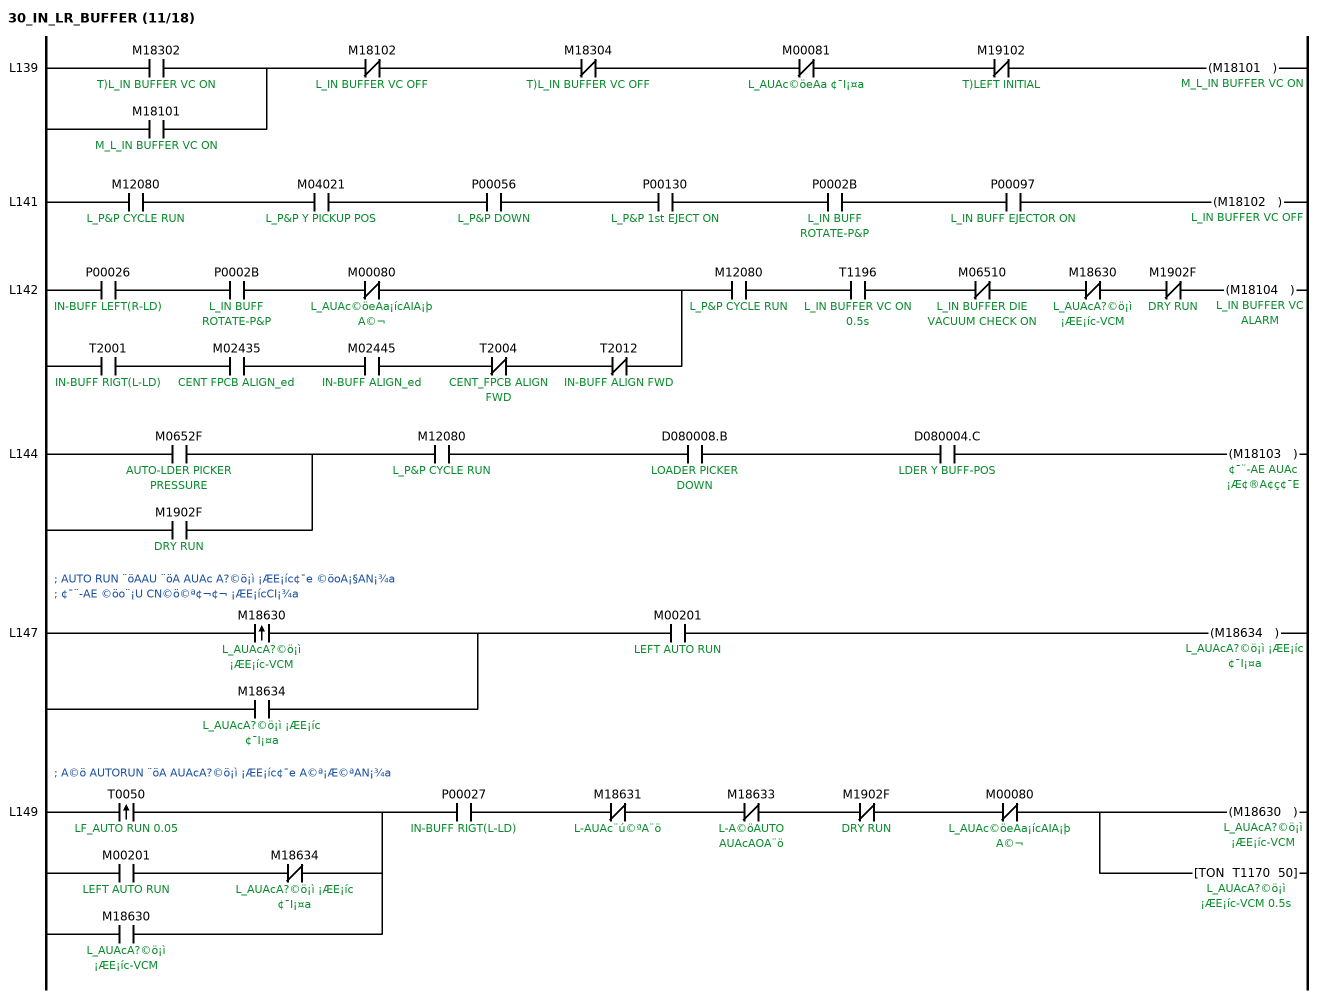
[picture p216: 30_IN_LR_BUFFER rungs L139-L149]
; L139
LOAD      M18302	// T)L_IN BUFFER VC ON
OR        M18101	// M_L_IN BUFFER VC ON
AND NOT   M18102	// L_IN BUFFER VC OFF
AND NOT   M18304	// T)L_IN BUFFER VC OFF
AND NOT   M00081	// L_AUAc©öeAa ¢¯I¡¤a
AND NOT   M19102	// T)LEFT INITIAL
OUT       M18101	// M_L_IN BUFFER VC ON
; L141
LOAD      M12080	// L_P&P CYCLE RUN
AND       M04021	// L_P&P Y PICKUP POS
AND       P00056	// L_P&P DOWN
AND       P00130	// L_P&P 1st EJECT ON
AND       P0002B	// L_IN BUFF ROTATE-P&P
AND       P00097	// L_IN BUFF EJECTOR ON
OUT       M18102	// L_IN BUFFER VC OFF
; L142
LOAD      P00026	// IN-BUFF LEFT(R-LD)
AND       P0002B	// L_IN BUFF ROTATE-P&P
AND NOT   M00080	// L_AUAc©öeAa¡ícAIA¡þA©¬
LOAD      T2001	// IN-BUFF RIGT(L-LD)
AND       M02435	// CENT FPCB ALIGN_ed
AND       M02445	// IN-BUFF ALIGN_ed
AND NOT   T2004	// CENT_FPCB ALIGN FWD
AND NOT   T2012	// IN-BUFF ALIGN FWD
OR LOAD
AND       M12080	// L_P&P CYCLE RUN
AND       T1196	// L_IN BUFFER VC ON 0.5s
AND NOT   M06510	// L_IN BUFFER DIE VACUUM CHECK ON
AND NOT   M18630	// L_AUAcA?©ö¡ì ¡ÆE¡íc-VCM
AND NOT   M1902F	// DRY RUN
OUT       M18104	// L_IN BUFFER VC ALARM
; L144
LOAD      M0652F	// AUTO-LDER PICKER PRESSURE
OR        M1902F	// DRY RUN
AND       M12080	// L_P&P CYCLE RUN
AND       D080008.B	// LOADER PICKER DOWN
AND       D080004.C	// LDER Y BUFF-POS
OUT       M18103	// ¢¯¨­AE AUAc ¡Æ¢®A¢ç¢¯E
// AUTO RUN ¨öAAU ¨öA AUAc A?©ö¡ì ¡ÆE¡íc¢¯e ©öoA¡§AN¡¾a
; L147
LOADP     M18630	// L_AUAcA?©ö¡ì ¡ÆE¡íc-VCM
OR        M18634	// L_AUAcA?©ö¡ì ¡ÆE¡íc ¢¯I¡¤a
AND       M00201	// LEFT AUTO RUN
OUT       M18634	// L_AUAcA?©ö¡ì ¡ÆE¡íc ¢¯I¡¤a
// output comment: ¢¯¨­AE ©öo¨¡U CN©ö©ª¢¬¢¬ ¡ÆE¡ícCI¡¾a
; L149
LOADP     T0050	// LF_AUTO RUN 0.05
LOAD      M00201	// LEFT AUTO RUN
AND NOT   M18634	// L_AUAcA?©ö¡ì ¡ÆE¡íc ¢¯I¡¤a
OR LOAD
OR        M18630	// L_AUAcA?©ö¡ì ¡ÆE¡íc-VCM
AND       P00027	// IN-BUFF RIGT(L-LD)
AND NOT   M18631	// L-AUAc¨ú©ªA¨ö
AND NOT   M18633	// L-A©öAUTO AUAcAOA¨ö
AND NOT   M1902F	// DRY RUN
AND NOT   M00080	// L_AUAc©öeAa¡ícAIA¡þA©¬
OUT       M18630	// L_AUAcA?©ö¡ì ¡ÆE¡íc-VCM
TON       T1170 50	// L_AUAcA?©ö¡ì ¡ÆE¡íc-VCM 0.5s
// output comment: A©ö AUTORUN ¨öA AUAcA?©ö¡ì ¡ÆE¡íc¢¯e A©ª¡Æ©ªAN¡¾a

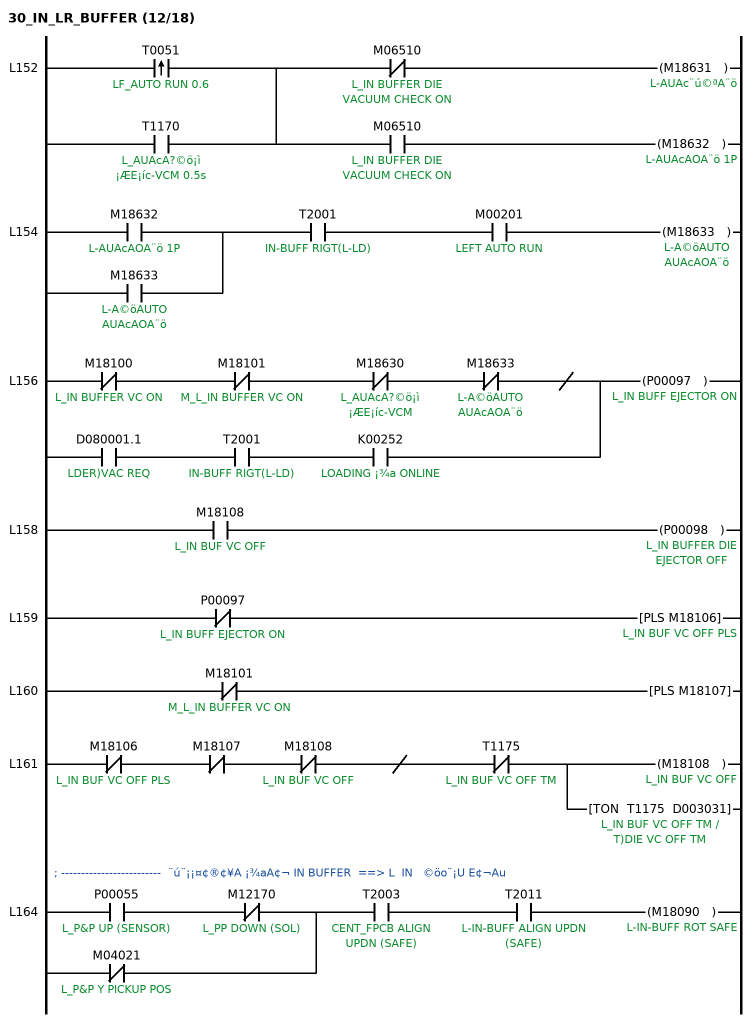
; L152
LOADP     T0051	// LF_AUTO RUN 0.6
OR        T1170	// L_AUAcA?©ö¡ì ¡ÆE¡íc-VCM 0.5s
MPUSH
AND NOT   M06510	// L_IN BUFFER DIE VACUUM CHECK ON
OUT       M18631	// L-AUAc¨ú©ªA¨ö
MPOP
AND       M06510	// L_IN BUFFER DIE VACUUM CHECK ON
OUT       M18632	// L-AUAcAOA¨ö 1P
; L154
LOAD      M18632	// L-AUAcAOA¨ö 1P
OR        M18633	// L-A©öAUTO AUAcAOA¨ö
AND       T2001	// IN-BUFF RIGT(L-LD)
AND       M00201	// LEFT AUTO RUN
OUT       M18633	// L-A©öAUTO AUAcAOA¨ö
; L156
LOAD NOT  M18100	// L_IN BUFFER VC ON
AND NOT   M18101	// M_L_IN BUFFER VC ON
AND NOT   M18630	// L_AUAcA?©ö¡ì ¡ÆE¡íc-VCM
AND NOT   M18633	// L-A©öAUTO AUAcAOA¨ö
NOT
LOAD      D080001.1	// LDER)VAC REQ
AND       T2001	// IN-BUFF RIGT(L-LD)
AND       K00252	// LOADING ¡¾a ONLINE
OR LOAD
OUT       P00097	// L_IN BUFF EJECTOR ON
; L158
LOAD      M18108	// L_IN BUF VC OFF
OUT       P00098	// L_IN BUFFER DIE EJECTOR OFF
; L159
LOAD NOT  P00097	// L_IN BUFF EJECTOR ON
OUTP      M18106	// L_IN BUF VC OFF PLS
; L160
LOAD NOT  M18101	// M_L_IN BUFFER VC ON
OUTP      M18107
; L161
LOAD NOT  M18106	// L_IN BUF VC OFF PLS
AND NOT   M18107
AND NOT   M18108	// L_IN BUF VC OFF
NOT
AND NOT   T1175	// L_IN BUF VC OFF TM
OUT       M18108	// L_IN BUF VC OFF
TON       T1175 D003031	// L_IN BUF VC OFF TM / T)DIE VC OFF TM
// -------------------------  ¨ú¨¡¡¤¢®¢¥A ¡¾aA¢¬ IN BUFFER  ==> L  IN   ©öo¨¡U E¢¬Au
; L164
LOAD      P00055	// L_P&P UP (SENSOR)
AND NOT   M12170	// L_PP DOWN (SOL)
OR NOT    M04021	// L_P&P Y PICKUP POS
AND       T2003	// CENT_FPCB ALIGN UPDN (SAFE)
AND       T2011	// L-IN-BUFF ALIGN UPDN (SAFE)
OUT       M18090	// L-IN-BUFF ROT SAFE

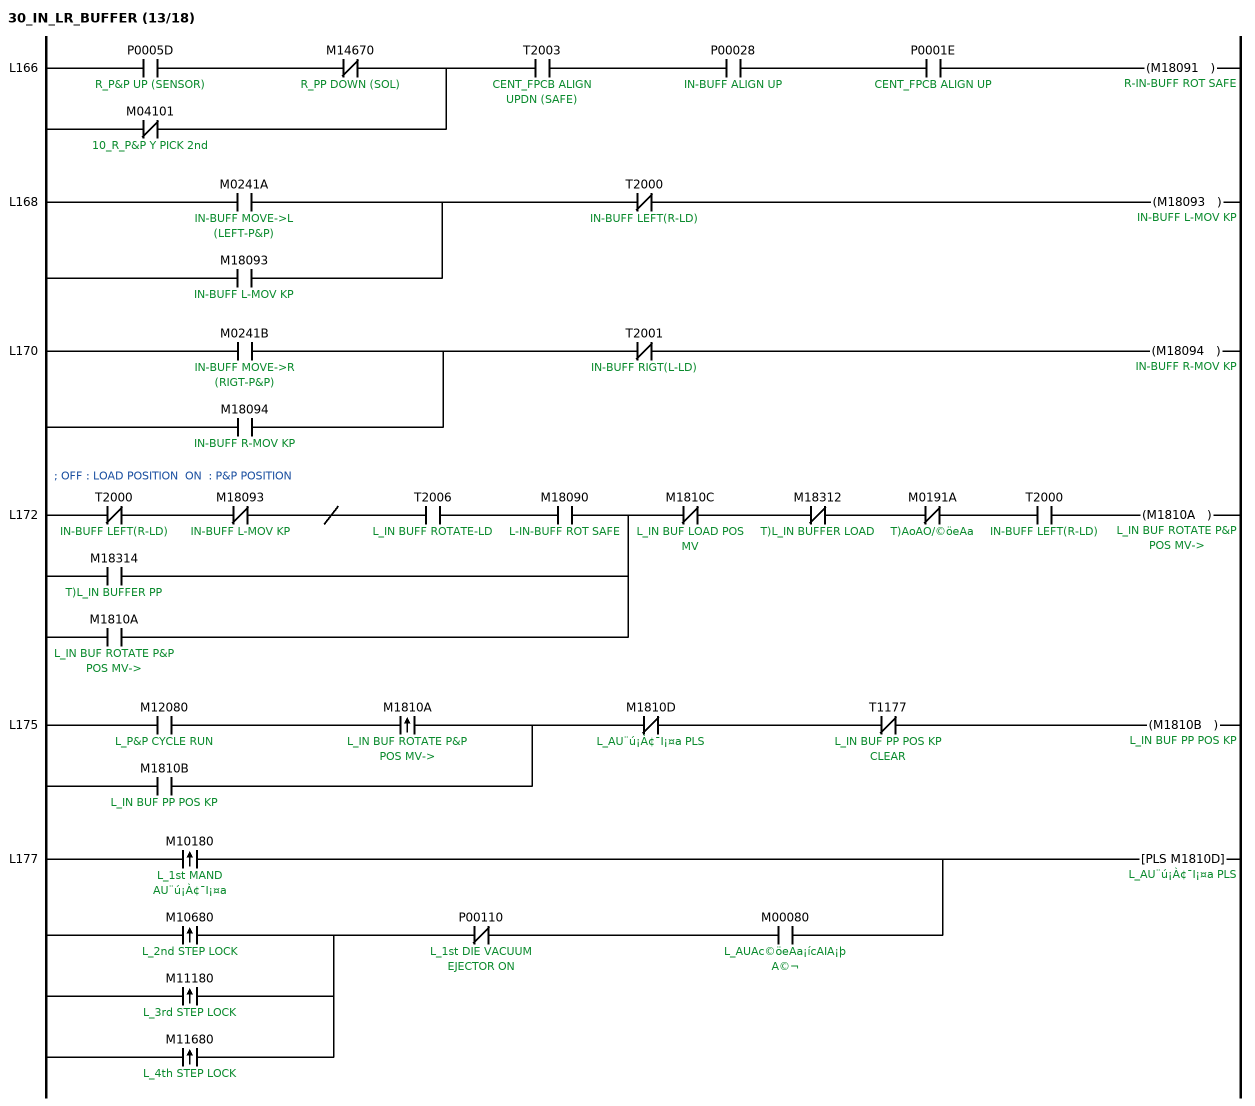
; L166
LOAD      P0005D	// R_P&P UP (SENSOR)
AND NOT   M14670	// R_PP DOWN (SOL)
OR NOT    M04101	// 10_R_P&P Y PICK 2nd
AND       T2003	// CENT_FPCB ALIGN UPDN (SAFE)
AND       P00028	// IN-BUFF ALIGN UP
AND       P0001E	// CENT_FPCB ALIGN UP
OUT       M18091	// R-IN-BUFF ROT SAFE
; L168
LOAD      M0241A	// IN-BUFF MOVE->L (LEFT-P&P)
OR        M18093	// IN-BUFF L-MOV KP
AND NOT   T2000	// IN-BUFF LEFT(R-LD)
OUT       M18093	// IN-BUFF L-MOV KP
; L170
LOAD      M0241B	// IN-BUFF MOVE->R (RIGT-P&P)
OR        M18094	// IN-BUFF R-MOV KP
AND NOT   T2001	// IN-BUFF RIGT(L-LD)
OUT       M18094	// IN-BUFF R-MOV KP
; L172
LOAD NOT  T2000	// IN-BUFF LEFT(R-LD)
AND NOT   M18093	// IN-BUFF L-MOV KP
NOT
AND       T2006	// L_IN BUFF ROTATE-LD
AND       M18090	// L-IN-BUFF ROT SAFE
OR        M18314	// T)L_IN BUFFER PP
OR        M1810A	// L_IN BUF ROTATE P&P POS MV->
AND NOT   M1810C	// L_IN BUF LOAD POS MV
AND NOT   M18312	// T)L_IN BUFFER LOAD
AND NOT   M0191A	// T)AoAO/©öeAa
AND       T2000	// IN-BUFF LEFT(R-LD)
OUT       M1810A	// L_IN BUF ROTATE P&P POS MV->
// output comment: OFF : LOAD POSITION  ON  : P&P POSITION
; L175
LOAD      M12080	// L_P&P CYCLE RUN
ANDP      M1810A	// L_IN BUF ROTATE P&P POS MV->
OR        M1810B	// L_IN BUF PP POS KP
AND NOT   M1810D	// L_AU¨ú¡À¢¯I¡¤a PLS
AND NOT   T1177	// L_IN BUF PP POS KP CLEAR
OUT       M1810B	// L_IN BUF PP POS KP
; L177
LOADP     M10180	// L_1st MAND AU¨ú¡À¢¯I¡¤a
LOADP     M10680	// L_2nd STEP LOCK
ORP       M11180	// L_3rd STEP LOCK
ORP       M11680	// L_4th STEP LOCK
AND NOT   P00110	// L_1st DIE VACUUM EJECTOR ON
AND       M00080	// L_AUAc©öeAa¡ícAIA¡þA©¬
OR LOAD
OUTP      M1810D	// L_AU¨ú¡À¢¯I¡¤a PLS

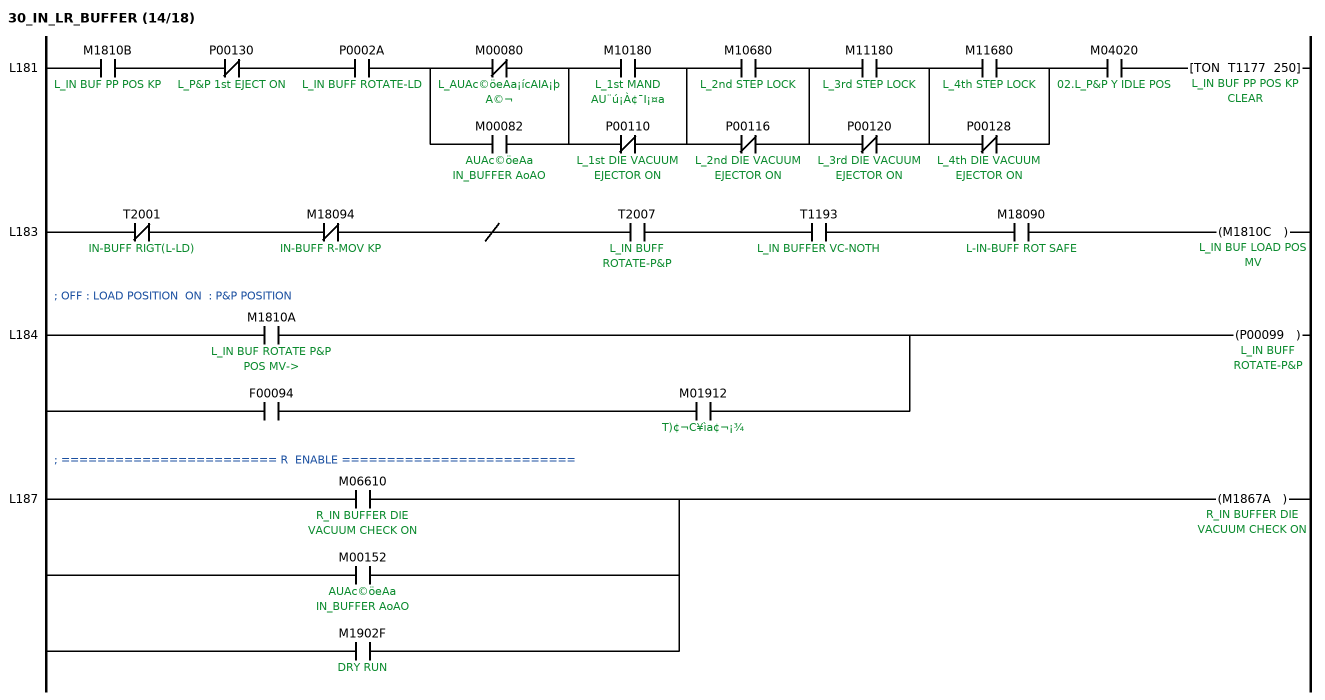
; L181
LOAD      M1810B	// L_IN BUF PP POS KP
AND NOT   P00130	// L_P&P 1st EJECT ON
AND       P0002A	// L_IN BUFF ROTATE-LD
LOAD NOT  M00080	// L_AUAc©öeAa¡ícAIA¡þA©¬
OR        M00082	// AUAc©öeAa IN_BUFFER AoAO 
AND LOAD
LOAD      M10180	// L_1st MAND AU¨ú¡À¢¯I¡¤a
OR NOT    P00110	// L_1st DIE VACUUM EJECTOR ON
AND LOAD
LOAD      M10680	// L_2nd STEP LOCK
OR NOT    P00116	// L_2nd DIE VACUUM EJECTOR ON
AND LOAD
LOAD      M11180	// L_3rd STEP LOCK
OR NOT    P00120	// L_3rd DIE VACUUM EJECTOR ON
AND LOAD
LOAD      M11680	// L_4th STEP LOCK
OR NOT    P00128	// L_4th DIE VACUUM EJECTOR ON
AND LOAD
AND       M04020	// 02.L_P&P Y IDLE POS
TON       T1177 250	// L_IN BUF PP POS KP CLEAR
; L183
LOAD NOT  T2001	// IN-BUFF RIGT(L-LD)
AND NOT   M18094	// IN-BUFF R-MOV KP
NOT
AND       T2007	// L_IN BUFF ROTATE-P&P
AND       T1193	// L_IN BUFFER VC-NOTH
AND       M18090	// L-IN-BUFF ROT SAFE
OUT       M1810C	// L_IN BUF LOAD POS MV
; L184
LOAD      M1810A	// L_IN BUF ROTATE P&P POS MV->
LOAD      F00094
AND       M01912	// T)¢¬C¥ìa¢¬¡¾
OR LOAD
OUT       P00099	// L_IN BUFF ROTATE-P&P
// output comment: OFF : LOAD POSITION  ON  : P&P POSITION
// ======================== R  ENABLE ==========================
; L187
LOAD      M06610	// R_IN BUFFER DIE VACUUM CHECK ON
OR        M00152	// AUAc©öeAa IN_BUFFER AoAO 
OR        M1902F	// DRY RUN
OUT       M1867A	// R_IN BUFFER DIE VACUUM CHECK ON

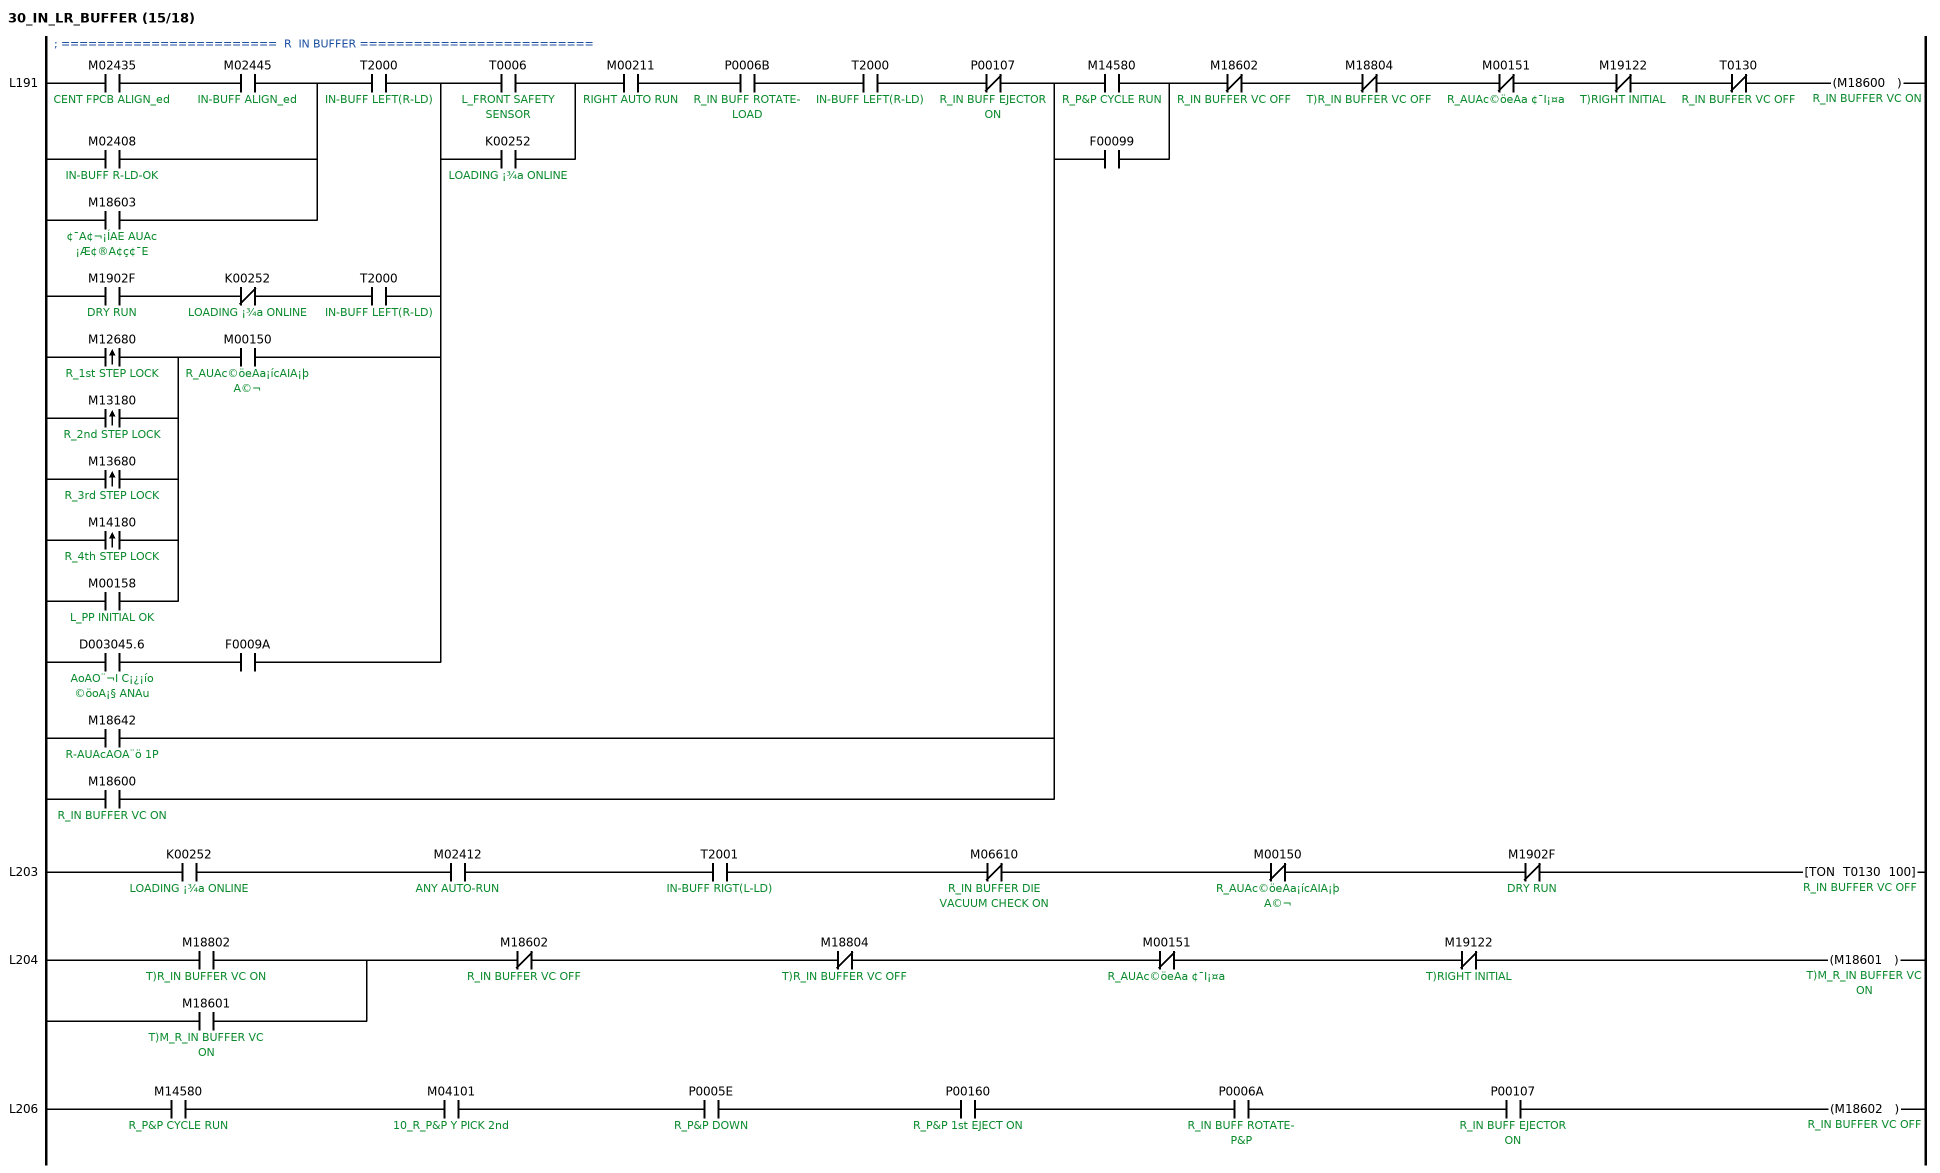
// ========================  R  IN BUFFER ==========================
; L191
LOAD      M02435	// CENT FPCB ALIGN_ed
AND       M02445	// IN-BUFF ALIGN_ed
OR        M02408	// IN-BUFF R-LD-OK
OR        M18603	// ¢¯A¢¬¡ÍAE AUAc ¡Æ¢®A¢ç¢¯E
AND       T2000	// IN-BUFF LEFT(R-LD)
LOAD      M1902F	// DRY RUN
AND NOT   K00252	// LOADING ¡¾a ONLINE
AND       T2000	// IN-BUFF LEFT(R-LD)
OR LOAD
LOADP     M12680	// R_1st STEP LOCK
ORP       M13180	// R_2nd STEP LOCK
ORP       M13680	// R_3rd STEP LOCK
ORP       M14180	// R_4th STEP LOCK
OR        M00158	// L_PP INITIAL OK
AND       M00150	// R_AUAc©öeAa¡ícAIA¡þA©¬
OR LOAD
LOAD      D003045.6	// AoAO¨¬I C¡¿¡ío ©öoA¡§ ANAu
AND       F0009A
OR LOAD
LOAD      T0006	// L_FRONT SAFETY SENSOR
OR        K00252	// LOADING ¡¾a ONLINE
AND LOAD
AND       M00211	// RIGHT AUTO RUN
AND       P0006B	// R_IN BUFF ROTATE- LOAD
AND       T2000	// IN-BUFF LEFT(R-LD)
AND NOT   P00107	// R_IN BUFF EJECTOR ON
OR        M18642	// R-AUAcAOA¨ö 1P
OR        M18600	// R_IN BUFFER VC ON
LOAD      M14580	// R_P&P CYCLE RUN
OR        F00099
AND LOAD
AND NOT   M18602	// R_IN BUFFER VC OFF
AND NOT   M18804	// T)R_IN BUFFER VC OFF
AND NOT   M00151	// R_AUAc©öeAa ¢¯I¡¤a
AND NOT   M19122	// T)RIGHT INITIAL
AND NOT   T0130	// R_IN BUFFER VC OFF
OUT       M18600	// R_IN BUFFER VC ON
; L203
LOAD      K00252	// LOADING ¡¾a ONLINE
AND       M02412	// ANY AUTO-RUN
AND       T2001	// IN-BUFF RIGT(L-LD)
AND NOT   M06610	// R_IN BUFFER DIE VACUUM CHECK ON
AND NOT   M00150	// R_AUAc©öeAa¡ícAIA¡þA©¬
AND NOT   M1902F	// DRY RUN
TON       T0130 100	// R_IN BUFFER VC OFF
; L204
LOAD      M18802	// T)R_IN BUFFER VC ON
OR        M18601	// T)M_R_IN BUFFER VC ON
AND NOT   M18602	// R_IN BUFFER VC OFF
AND NOT   M18804	// T)R_IN BUFFER VC OFF
AND NOT   M00151	// R_AUAc©öeAa ¢¯I¡¤a
AND NOT   M19122	// T)RIGHT INITIAL
OUT       M18601	// T)M_R_IN BUFFER VC ON
; L206
LOAD      M14580	// R_P&P CYCLE RUN
AND       M04101	// 10_R_P&P Y PICK 2nd
AND       P0005E	// R_P&P DOWN
AND       P00160	// R_P&P 1st EJECT ON
AND       P0006A	// R_IN BUFF ROTATE- P&P
AND       P00107	// R_IN BUFF EJECTOR ON
OUT       M18602	// R_IN BUFFER VC OFF

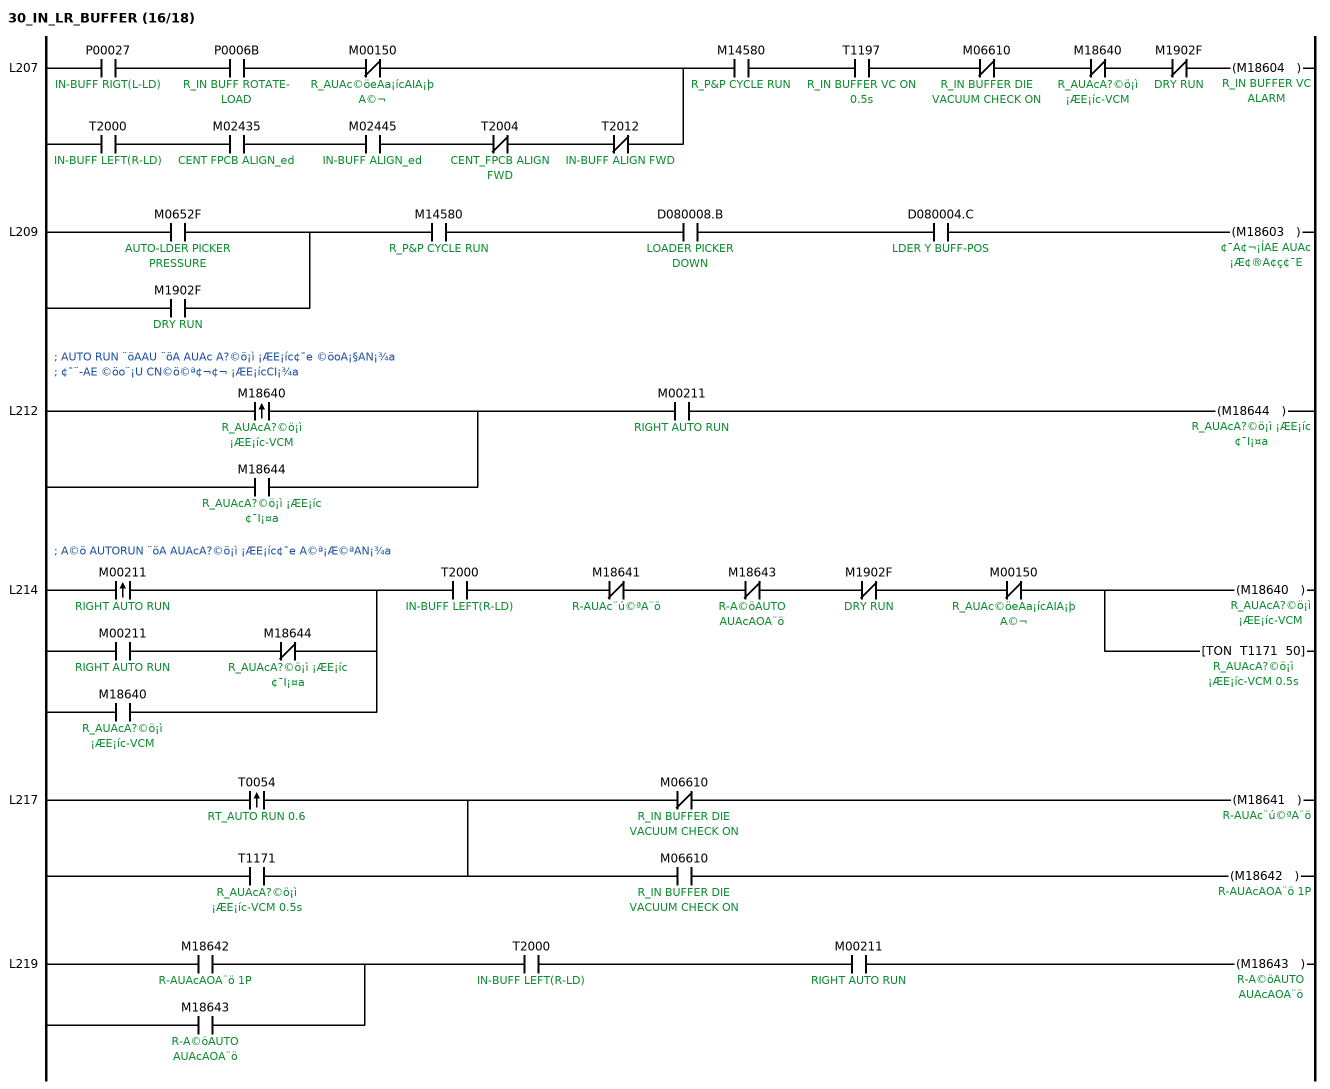
; L207
LOAD      P00027	// IN-BUFF RIGT(L-LD)
AND       P0006B	// R_IN BUFF ROTATE- LOAD
AND NOT   M00150	// R_AUAc©öeAa¡ícAIA¡þA©¬
LOAD      T2000	// IN-BUFF LEFT(R-LD)
AND       M02435	// CENT FPCB ALIGN_ed
AND       M02445	// IN-BUFF ALIGN_ed
AND NOT   T2004	// CENT_FPCB ALIGN FWD
AND NOT   T2012	// IN-BUFF ALIGN FWD
OR LOAD
AND       M14580	// R_P&P CYCLE RUN
AND       T1197	// R_IN BUFFER VC ON 0.5s
AND NOT   M06610	// R_IN BUFFER DIE VACUUM CHECK ON
AND NOT   M18640	// R_AUAcA?©ö¡ì ¡ÆE¡íc-VCM
AND NOT   M1902F	// DRY RUN
OUT       M18604	// R_IN BUFFER VC ALARM
; L209
LOAD      M0652F	// AUTO-LDER PICKER PRESSURE
OR        M1902F	// DRY RUN
AND       M14580	// R_P&P CYCLE RUN
AND       D080008.B	// LOADER PICKER DOWN
AND       D080004.C	// LDER Y BUFF-POS
OUT       M18603	// ¢¯A¢¬¡ÍAE AUAc ¡Æ¢®A¢ç¢¯E
// AUTO RUN ¨öAAU ¨öA AUAc A?©ö¡ì ¡ÆE¡íc¢¯e ©öoA¡§AN¡¾a
; L212
LOADP     M18640	// R_AUAcA?©ö¡ì ¡ÆE¡íc-VCM
OR        M18644	// R_AUAcA?©ö¡ì ¡ÆE¡íc ¢¯I¡¤a
AND       M00211	// RIGHT AUTO RUN
OUT       M18644	// R_AUAcA?©ö¡ì ¡ÆE¡íc ¢¯I¡¤a
// output comment: ¢¯¨­AE ©öo¨¡U CN©ö©ª¢¬¢¬ ¡ÆE¡ícCI¡¾a
; L214
LOADP     M00211	// RIGHT AUTO RUN
LOAD      M00211	// RIGHT AUTO RUN
AND NOT   M18644	// R_AUAcA?©ö¡ì ¡ÆE¡íc ¢¯I¡¤a
OR LOAD
OR        M18640	// R_AUAcA?©ö¡ì ¡ÆE¡íc-VCM
AND       T2000	// IN-BUFF LEFT(R-LD)
AND NOT   M18641	// R-AUAc¨ú©ªA¨ö
AND NOT   M18643	// R-A©öAUTO AUAcAOA¨ö
AND NOT   M1902F	// DRY RUN
AND NOT   M00150	// R_AUAc©öeAa¡ícAIA¡þA©¬
OUT       M18640	// R_AUAcA?©ö¡ì ¡ÆE¡íc-VCM
TON       T1171 50	// R_AUAcA?©ö¡ì ¡ÆE¡íc-VCM 0.5s
// output comment: A©ö AUTORUN ¨öA AUAcA?©ö¡ì ¡ÆE¡íc¢¯e A©ª¡Æ©ªAN¡¾a
; L217
LOADP     T0054	// RT_AUTO RUN 0.6
OR        T1171	// R_AUAcA?©ö¡ì ¡ÆE¡íc-VCM 0.5s
MPUSH
AND NOT   M06610	// R_IN BUFFER DIE VACUUM CHECK ON
OUT       M18641	// R-AUAc¨ú©ªA¨ö
MPOP
AND       M06610	// R_IN BUFFER DIE VACUUM CHECK ON
OUT       M18642	// R-AUAcAOA¨ö 1P
; L219
LOAD      M18642	// R-AUAcAOA¨ö 1P
OR        M18643	// R-A©öAUTO AUAcAOA¨ö
AND       T2000	// IN-BUFF LEFT(R-LD)
AND       M00211	// RIGHT AUTO RUN
OUT       M18643	// R-A©öAUTO AUAcAOA¨ö

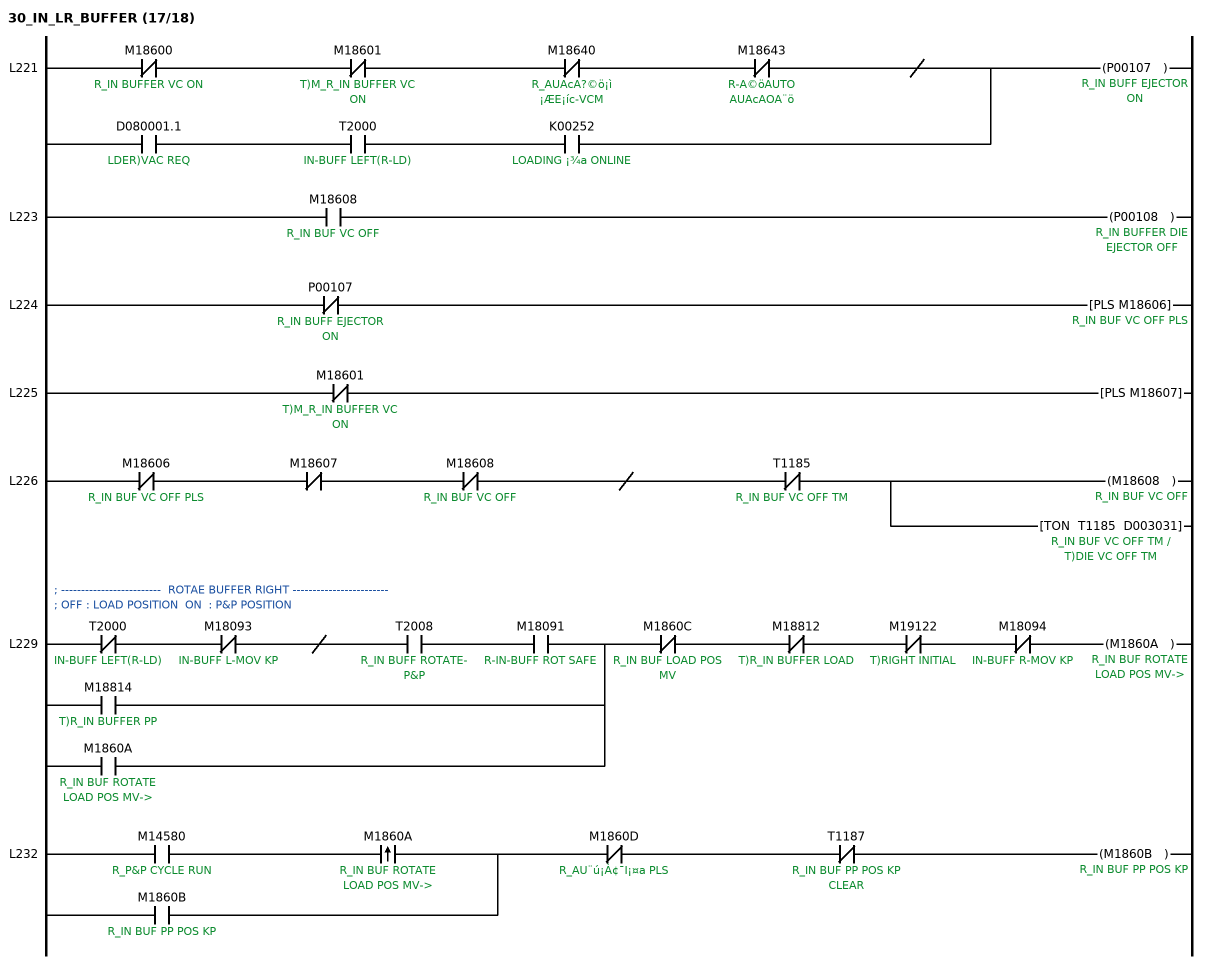
; L221
LOAD NOT  M18600	// R_IN BUFFER VC ON
AND NOT   M18601	// T)M_R_IN BUFFER VC ON
AND NOT   M18640	// R_AUAcA?©ö¡ì ¡ÆE¡íc-VCM
AND NOT   M18643	// R-A©öAUTO AUAcAOA¨ö
NOT
LOAD      D080001.1	// LDER)VAC REQ
AND       T2000	// IN-BUFF LEFT(R-LD)
AND       K00252	// LOADING ¡¾a ONLINE
OR LOAD
OUT       P00107	// R_IN BUFF EJECTOR ON
; L223
LOAD      M18608	// R_IN BUF VC OFF
OUT       P00108	// R_IN BUFFER DIE EJECTOR OFF
; L224
LOAD NOT  P00107	// R_IN BUFF EJECTOR ON
OUTP      M18606	// R_IN BUF VC OFF PLS
; L225
LOAD NOT  M18601	// T)M_R_IN BUFFER VC ON
OUTP      M18607
; L226
LOAD NOT  M18606	// R_IN BUF VC OFF PLS
AND NOT   M18607
AND NOT   M18608	// R_IN BUF VC OFF
NOT
AND NOT   T1185	// R_IN BUF VC OFF TM
OUT       M18608	// R_IN BUF VC OFF
TON       T1185 D003031	// R_IN BUF VC OFF TM / T)DIE VC OFF TM
// -------------------------  ROTAE BUFFER RIGHT ------------------------
; L229
LOAD NOT  T2000	// IN-BUFF LEFT(R-LD)
AND NOT   M18093	// IN-BUFF L-MOV KP
NOT
AND       T2008	// R_IN BUFF ROTATE- P&P
AND       M18091	// R-IN-BUFF ROT SAFE
OR        M18814	// T)R_IN BUFFER PP
OR        M1860A	// R_IN BUF ROTATE LOAD POS MV->
AND NOT   M1860C	// R_IN BUF LOAD POS MV
AND NOT   M18812	// T)R_IN BUFFER LOAD
AND NOT   M19122	// T)RIGHT INITIAL
AND NOT   M18094	// IN-BUFF R-MOV KP
OUT       M1860A	// R_IN BUF ROTATE LOAD POS MV->
// output comment: OFF : LOAD POSITION  ON  : P&P POSITION
; L232
LOAD      M14580	// R_P&P CYCLE RUN
ANDP      M1860A	// R_IN BUF ROTATE LOAD POS MV->
OR        M1860B	// R_IN BUF PP POS KP
AND NOT   M1860D	// R_AU¨ú¡À¢¯I¡¤a PLS
AND NOT   T1187	// R_IN BUF PP POS KP CLEAR
OUT       M1860B	// R_IN BUF PP POS KP

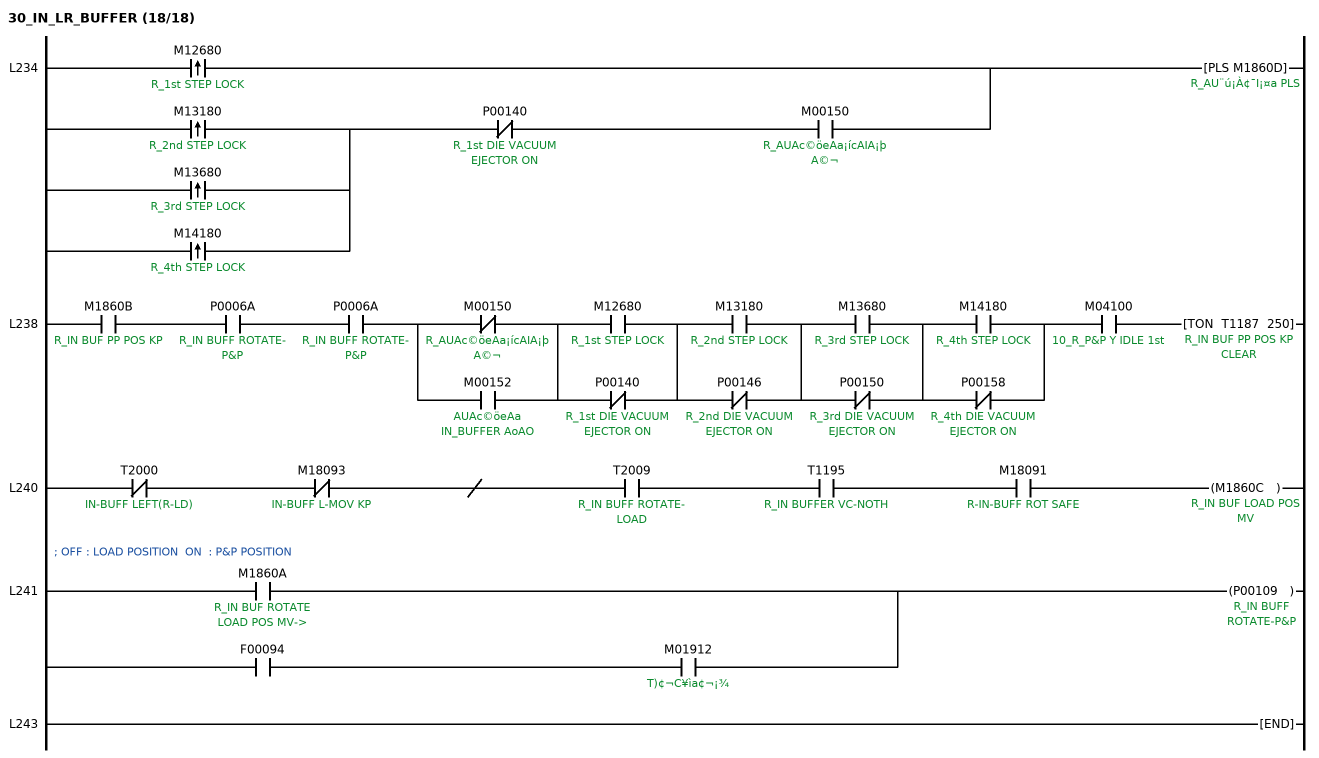
; L234
LOADP     M12680	// R_1st STEP LOCK
LOADP     M13180	// R_2nd STEP LOCK
ORP       M13680	// R_3rd STEP LOCK
ORP       M14180	// R_4th STEP LOCK
AND NOT   P00140	// R_1st DIE VACUUM EJECTOR ON
AND       M00150	// R_AUAc©öeAa¡ícAIA¡þA©¬
OR LOAD
OUTP      M1860D	// R_AU¨ú¡À¢¯I¡¤a PLS
; L238
LOAD      M1860B	// R_IN BUF PP POS KP
AND       P0006A	// R_IN BUFF ROTATE- P&P
AND       P0006A	// R_IN BUFF ROTATE- P&P
LOAD NOT  M00150	// R_AUAc©öeAa¡ícAIA¡þA©¬
OR        M00152	// AUAc©öeAa IN_BUFFER AoAO 
AND LOAD
LOAD      M12680	// R_1st STEP LOCK
OR NOT    P00140	// R_1st DIE VACUUM EJECTOR ON
AND LOAD
LOAD      M13180	// R_2nd STEP LOCK
OR NOT    P00146	// R_2nd DIE VACUUM EJECTOR ON
AND LOAD
LOAD      M13680	// R_3rd STEP LOCK
OR NOT    P00150	// R_3rd DIE VACUUM EJECTOR ON
AND LOAD
LOAD      M14180	// R_4th STEP LOCK
OR NOT    P00158	// R_4th DIE VACUUM EJECTOR ON
AND LOAD
AND       M04100	// 10_R_P&P Y IDLE 1st
TON       T1187 250	// R_IN BUF PP POS KP CLEAR
; L240
LOAD NOT  T2000	// IN-BUFF LEFT(R-LD)
AND NOT   M18093	// IN-BUFF L-MOV KP
NOT
AND       T2009	// R_IN BUFF ROTATE- LOAD
AND       T1195	// R_IN BUFFER VC-NOTH
AND       M18091	// R-IN-BUFF ROT SAFE
OUT       M1860C	// R_IN BUF LOAD POS MV
; L241
LOAD      M1860A	// R_IN BUF ROTATE LOAD POS MV->
LOAD      F00094
AND       M01912	// T)¢¬C¥ìa¢¬¡¾
OR LOAD
OUT       P00109	// R_IN BUFF ROTATE-P&P
// output comment: OFF : LOAD POSITION  ON  : P&P POSITION
; L243
END

PROGRAM 31_OUT_LR_BUFFER (task: ¨ö¨¬A¥ì CA¡¤I¡¾¡¿¡¤¡Í)

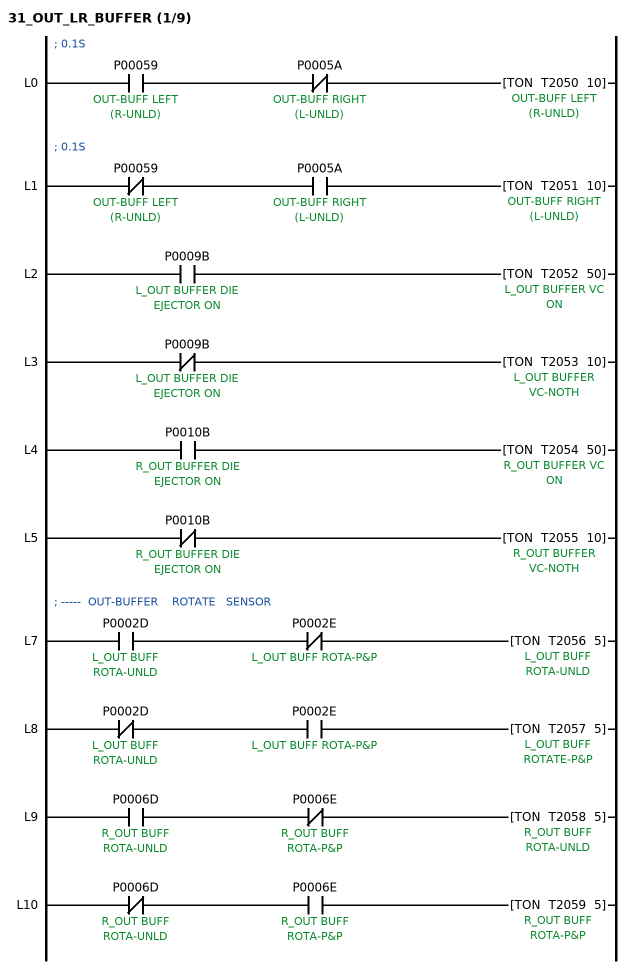
; L0
LOAD      P00059	// OUT-BUFF LEFT (R-UNLD)
AND NOT   P0005A	// OUT-BUFF RIGHT (L-UNLD)
TON       T2050 10	// OUT-BUFF LEFT (R-UNLD)
// output comment: 0.1S
; L1
LOAD NOT  P00059	// OUT-BUFF LEFT (R-UNLD)
AND       P0005A	// OUT-BUFF RIGHT (L-UNLD)
TON       T2051 10	// OUT-BUFF RIGHT (L-UNLD)
// output comment: 0.1S
; L2
LOAD      P0009B	// L_OUT BUFFER DIE EJECTOR ON
TON       T2052 50	// L_OUT BUFFER VC ON
; L3
LOAD NOT  P0009B	// L_OUT BUFFER DIE EJECTOR ON
TON       T2053 10	// L_OUT BUFFER VC-NOTH
; L4
LOAD      P0010B	// R_OUT BUFFER DIE EJECTOR ON
TON       T2054 50	// R_OUT BUFFER VC ON
; L5
LOAD NOT  P0010B	// R_OUT BUFFER DIE EJECTOR ON
TON       T2055 10	// R_OUT BUFFER VC-NOTH
// -----  OUT-BUFFER    ROTATE   SENSOR
; L7
LOAD      P0002D	// L_OUT BUFF ROTA-UNLD
AND NOT   P0002E	// L_OUT BUFF ROTA-P&P
TON       T2056 5	// L_OUT BUFF ROTA-UNLD
; L8
LOAD NOT  P0002D	// L_OUT BUFF ROTA-UNLD
AND       P0002E	// L_OUT BUFF ROTA-P&P
TON       T2057 5	// L_OUT BUFF ROTATE-P&P
; L9
LOAD      P0006D	// R_OUT BUFF ROTA-UNLD
AND NOT   P0006E	// R_OUT BUFF ROTA-P&P
TON       T2058 5	// R_OUT BUFF ROTA-UNLD
; L10
LOAD NOT  P0006D	// R_OUT BUFF ROTA-UNLD
AND       P0006E	// R_OUT BUFF ROTA-P&P
TON       T2059 5	// R_OUT BUFF ROTA-P&P

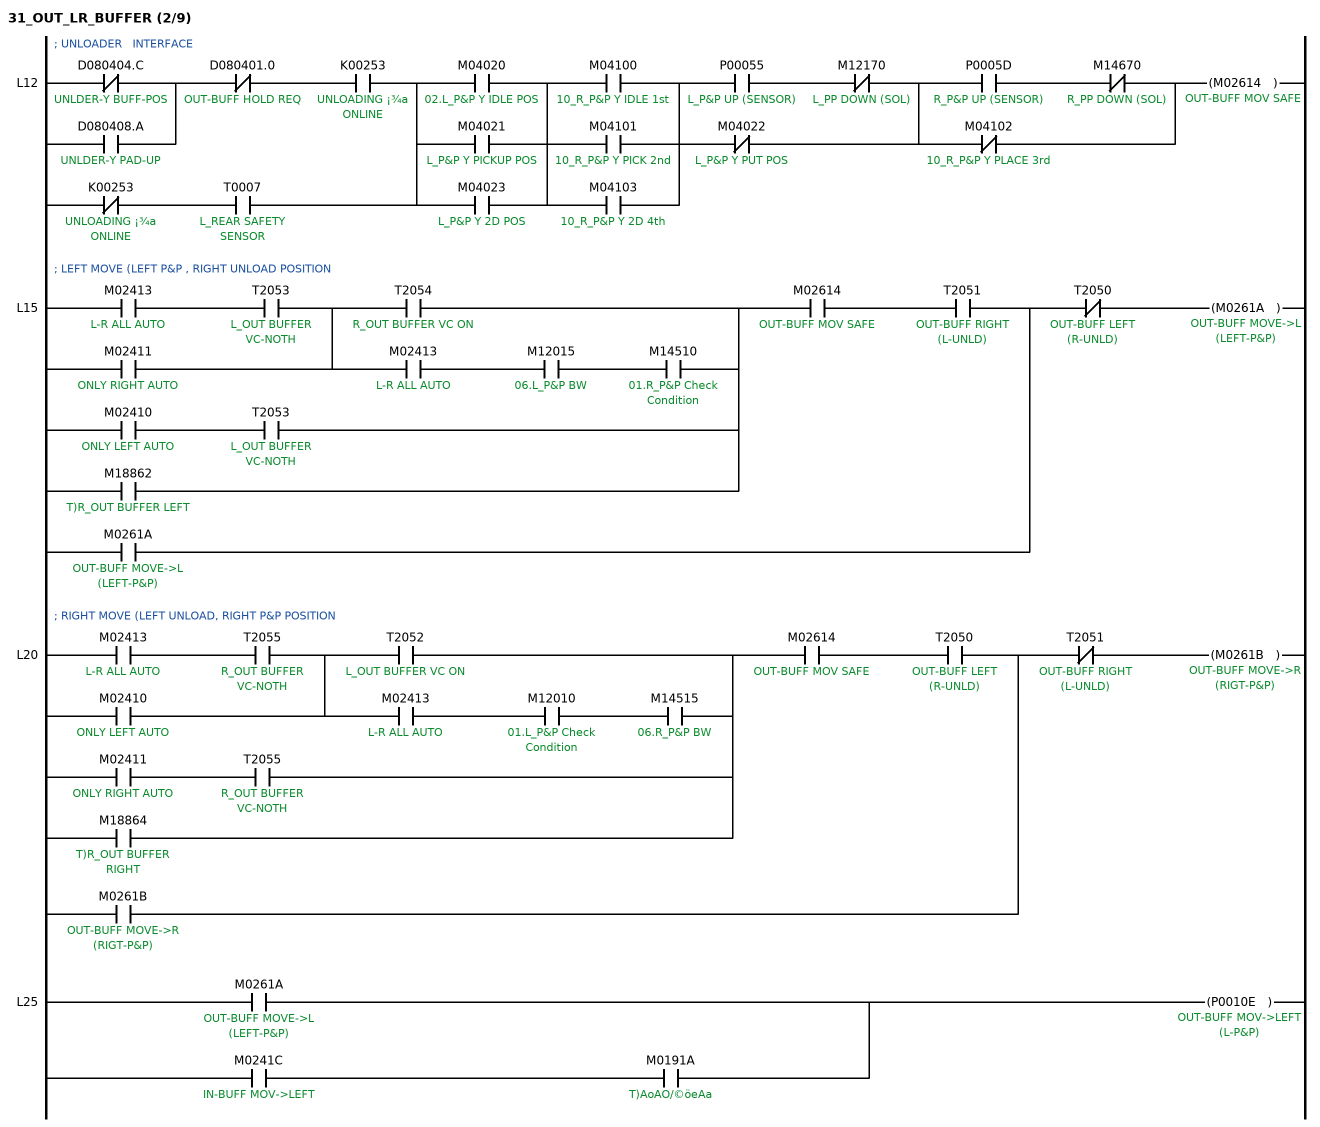
//  UNLOADER   INTERFACE
; L12
LOAD NOT  D080404.C	// UNLDER-Y BUFF-POS
OR        D080408.A	// UNLDER-Y PAD-UP
AND NOT   D080401.0	// OUT-BUFF HOLD REQ
AND       K00253	// UNLOADING ¡¾a ONLINE
LOAD NOT  K00253	// UNLOADING ¡¾a ONLINE
AND       T0007	// L_REAR SAFETY SENSOR
OR LOAD
LOAD      M04020	// 02.L_P&P Y IDLE POS
OR        M04021	// L_P&P Y PICKUP POS
OR        M04023	// L_P&P Y 2D POS
AND LOAD
LOAD      M04100	// 10_R_P&P Y IDLE 1st
OR        M04101	// 10_R_P&P Y PICK 2nd
OR        M04103	// 10_R_P&P Y 2D 4th
AND LOAD
LOAD      P00055	// L_P&P UP (SENSOR)
AND NOT   M12170	// L_PP DOWN (SOL)
OR NOT    M04022	// L_P&P Y PUT POS
AND LOAD
LOAD      P0005D	// R_P&P UP (SENSOR)
AND NOT   M14670	// R_PP DOWN (SOL)
OR NOT    M04102	// 10_R_P&P Y PLACE 3rd
AND LOAD
OUT       M02614	// OUT-BUFF MOV SAFE
; L15
LOAD      M02413	// L-R ALL AUTO
AND       T2053	// L_OUT BUFFER VC-NOTH
OR        M02411	// ONLY RIGHT AUTO
LOAD      T2054	// R_OUT BUFFER VC ON
LOAD      M02413	// L-R ALL AUTO
AND       M12015	// 06.L_P&P BW
AND       M14510	// 01.R_P&P Check Condition
OR LOAD
AND LOAD
LOAD      M02410	// ONLY LEFT AUTO
AND       T2053	// L_OUT BUFFER VC-NOTH
OR LOAD
OR        M18862	// T)R_OUT BUFFER LEFT
AND       M02614	// OUT-BUFF MOV SAFE
AND       T2051	// OUT-BUFF RIGHT (L-UNLD)
OR        M0261A	// OUT-BUFF MOVE->L (LEFT-P&P)
AND NOT   T2050	// OUT-BUFF LEFT (R-UNLD)
OUT       M0261A	// OUT-BUFF MOVE->L (LEFT-P&P)
// output comment: LEFT MOVE (LEFT P&P , RIGHT UNLOAD POSITION
; L20
LOAD      M02413	// L-R ALL AUTO
AND       T2055	// R_OUT BUFFER VC-NOTH
OR        M02410	// ONLY LEFT AUTO
LOAD      T2052	// L_OUT BUFFER VC ON
LOAD      M02413	// L-R ALL AUTO
AND       M12010	// 01.L_P&P Check Condition
AND       M14515	// 06.R_P&P BW
OR LOAD
AND LOAD
LOAD      M02411	// ONLY RIGHT AUTO
AND       T2055	// R_OUT BUFFER VC-NOTH
OR LOAD
OR        M18864	// T)R_OUT BUFFER RIGHT
AND       M02614	// OUT-BUFF MOV SAFE
AND       T2050	// OUT-BUFF LEFT (R-UNLD)
OR        M0261B	// OUT-BUFF MOVE->R (RIGT-P&P)
AND NOT   T2051	// OUT-BUFF RIGHT (L-UNLD)
OUT       M0261B	// OUT-BUFF MOVE->R (RIGT-P&P)
// output comment: RIGHT MOVE (LEFT UNLOAD, RIGHT P&P POSITION
; L25
LOAD      M0261A	// OUT-BUFF MOVE->L (LEFT-P&P)
LOAD      M0241C	// IN-BUFF MOV->LEFT
AND       M0191A	// T)AoAO/©öeAa
OR LOAD
OUT       P0010E	// OUT-BUFF MOV->LEFT (L-P&P)

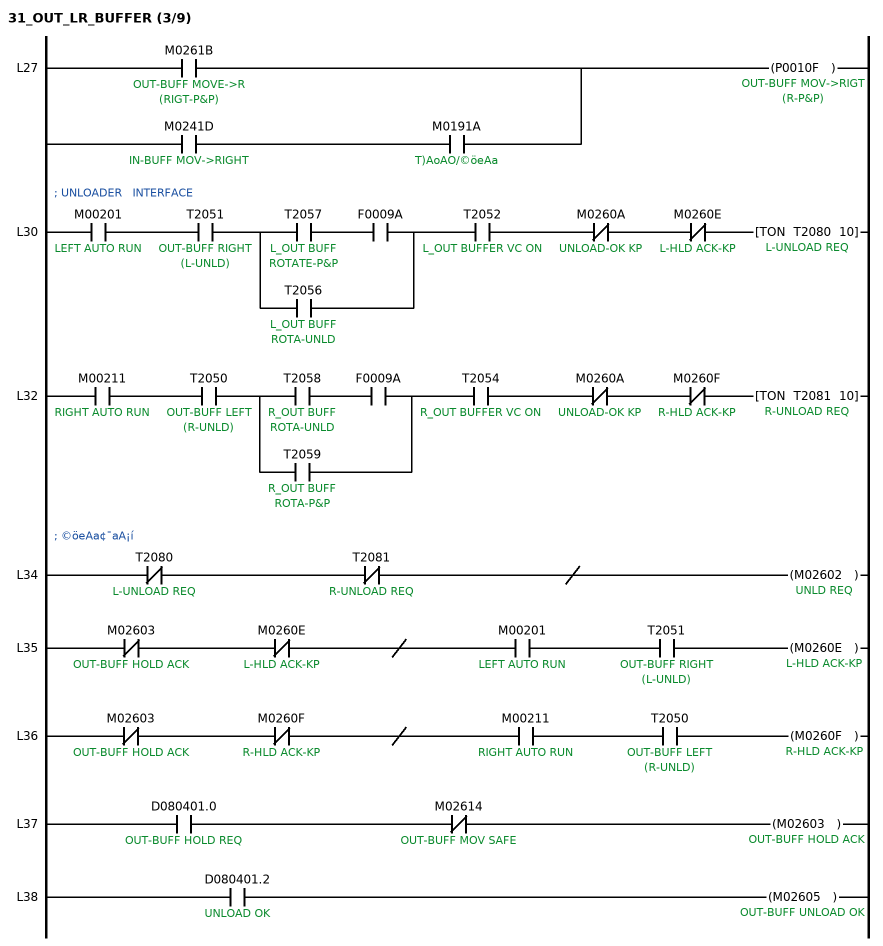
; L27
LOAD      M0261B	// OUT-BUFF MOVE->R (RIGT-P&P)
LOAD      M0241D	// IN-BUFF MOV->RIGHT
AND       M0191A	// T)AoAO/©öeAa
OR LOAD
OUT       P0010F	// OUT-BUFF MOV->RIGT (R-P&P)
//  UNLOADER   INTERFACE
; L30
LOAD      M00201	// LEFT AUTO RUN
AND       T2051	// OUT-BUFF RIGHT (L-UNLD)
LOAD      T2057	// L_OUT BUFF ROTATE-P&P
AND       F0009A
OR        T2056	// L_OUT BUFF ROTA-UNLD
AND LOAD
AND       T2052	// L_OUT BUFFER VC ON
AND NOT   M0260A	// UNLOAD-OK KP
AND NOT   M0260E	// L-HLD ACK-KP
TON       T2080 10	// L-UNLOAD REQ
; L32
LOAD      M00211	// RIGHT AUTO RUN
AND       T2050	// OUT-BUFF LEFT (R-UNLD)
LOAD      T2058	// R_OUT BUFF ROTA-UNLD
AND       F0009A
OR        T2059	// R_OUT BUFF ROTA-P&P
AND LOAD
AND       T2054	// R_OUT BUFFER VC ON
AND NOT   M0260A	// UNLOAD-OK KP
AND NOT   M0260F	// R-HLD ACK-KP
TON       T2081 10	// R-UNLOAD REQ
; L34
LOAD NOT  T2080	// L-UNLOAD REQ
AND NOT   T2081	// R-UNLOAD REQ
NOT
OUT       M02602	// UNLD REQ
// output comment: ©öeAa¢¯aA¡í
; L35
LOAD NOT  M02603	// OUT-BUFF HOLD ACK
AND NOT   M0260E	// L-HLD ACK-KP
NOT
AND       M00201	// LEFT AUTO RUN
AND       T2051	// OUT-BUFF RIGHT (L-UNLD)
OUT       M0260E	// L-HLD ACK-KP
; L36
LOAD NOT  M02603	// OUT-BUFF HOLD ACK
AND NOT   M0260F	// R-HLD ACK-KP
NOT
AND       M00211	// RIGHT AUTO RUN
AND       T2050	// OUT-BUFF LEFT (R-UNLD)
OUT       M0260F	// R-HLD ACK-KP
; L37
LOAD      D080401.0	// OUT-BUFF HOLD REQ
AND NOT   M02614	// OUT-BUFF MOV SAFE
OUT       M02603	// OUT-BUFF HOLD ACK
; L38
LOAD      D080401.2	// UNLOAD OK
OUT       M02605	// OUT-BUFF UNLOAD OK

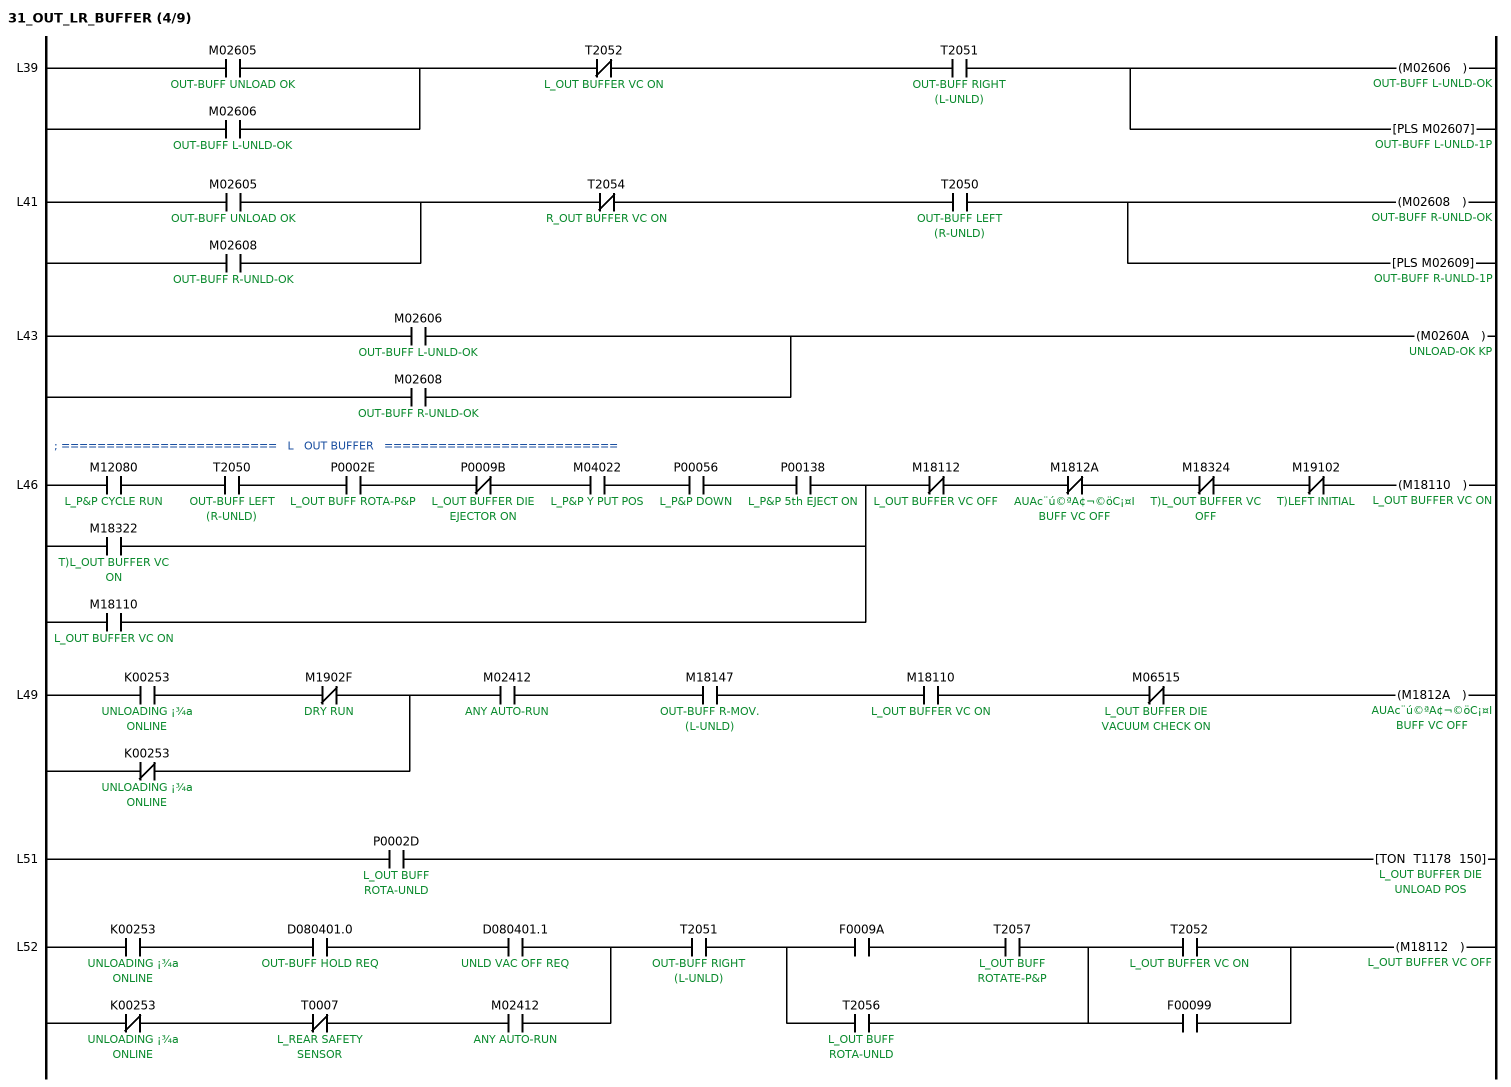
; L39
LOAD      M02605	// OUT-BUFF UNLOAD OK
OR        M02606	// OUT-BUFF L-UNLD-OK
AND NOT   T2052	// L_OUT BUFFER VC ON
AND       T2051	// OUT-BUFF RIGHT (L-UNLD)
OUT       M02606	// OUT-BUFF L-UNLD-OK
OUTP      M02607	// OUT-BUFF L-UNLD-1P
; L41
LOAD      M02605	// OUT-BUFF UNLOAD OK
OR        M02608	// OUT-BUFF R-UNLD-OK
AND NOT   T2054	// R_OUT BUFFER VC ON
AND       T2050	// OUT-BUFF LEFT (R-UNLD)
OUT       M02608	// OUT-BUFF R-UNLD-OK
OUTP      M02609	// OUT-BUFF R-UNLD-1P
; L43
LOAD      M02606	// OUT-BUFF L-UNLD-OK
OR        M02608	// OUT-BUFF R-UNLD-OK
OUT       M0260A	// UNLOAD-OK KP
// ========================   L   OUT BUFFER   ==========================
; L46
LOAD      M12080	// L_P&P CYCLE RUN
AND       T2050	// OUT-BUFF LEFT (R-UNLD)
AND       P0002E	// L_OUT BUFF ROTA-P&P
AND NOT   P0009B	// L_OUT BUFFER DIE EJECTOR ON
AND       M04022	// L_P&P Y PUT POS
AND       P00056	// L_P&P DOWN
AND       P00138	// L_P&P 5th EJECT ON
OR        M18322	// T)L_OUT BUFFER VC ON
OR        M18110	// L_OUT BUFFER VC ON
AND NOT   M18112	// L_OUT BUFFER VC OFF
AND NOT   M1812A	// AUAc¨ú©ªA¢¬©öC¡¤I BUFF VC OFF
AND NOT   M18324	// T)L_OUT BUFFER VC OFF
AND NOT   M19102	// T)LEFT INITIAL
OUT       M18110	// L_OUT BUFFER VC ON
; L49
LOAD      K00253	// UNLOADING ¡¾a ONLINE
AND NOT   M1902F	// DRY RUN
OR NOT    K00253	// UNLOADING ¡¾a ONLINE
AND       M02412	// ANY AUTO-RUN
AND       M18147	// OUT-BUFF R-MOV.  (L-UNLD)
AND       M18110	// L_OUT BUFFER VC ON
AND NOT   M06515	// L_OUT BUFFER DIE VACUUM CHECK ON
OUT       M1812A	// AUAc¨ú©ªA¢¬©öC¡¤I BUFF VC OFF
; L51
LOAD      P0002D	// L_OUT BUFF ROTA-UNLD
TON       T1178 150	// L_OUT BUFFER DIE UNLOAD POS
; L52
LOAD      K00253	// UNLOADING ¡¾a ONLINE
AND       D080401.0	// OUT-BUFF HOLD REQ
AND       D080401.1	// UNLD VAC OFF REQ
LOAD NOT  K00253	// UNLOADING ¡¾a ONLINE
AND NOT   T0007	// L_REAR SAFETY SENSOR
AND       M02412	// ANY AUTO-RUN
OR LOAD
AND       T2051	// OUT-BUFF RIGHT (L-UNLD)
LOAD      F0009A
AND       T2057	// L_OUT BUFF ROTATE-P&P
OR        T2056	// L_OUT BUFF ROTA-UNLD
AND LOAD
LOAD      T2052	// L_OUT BUFFER VC ON
OR        F00099
AND LOAD
OUT       M18112	// L_OUT BUFFER VC OFF

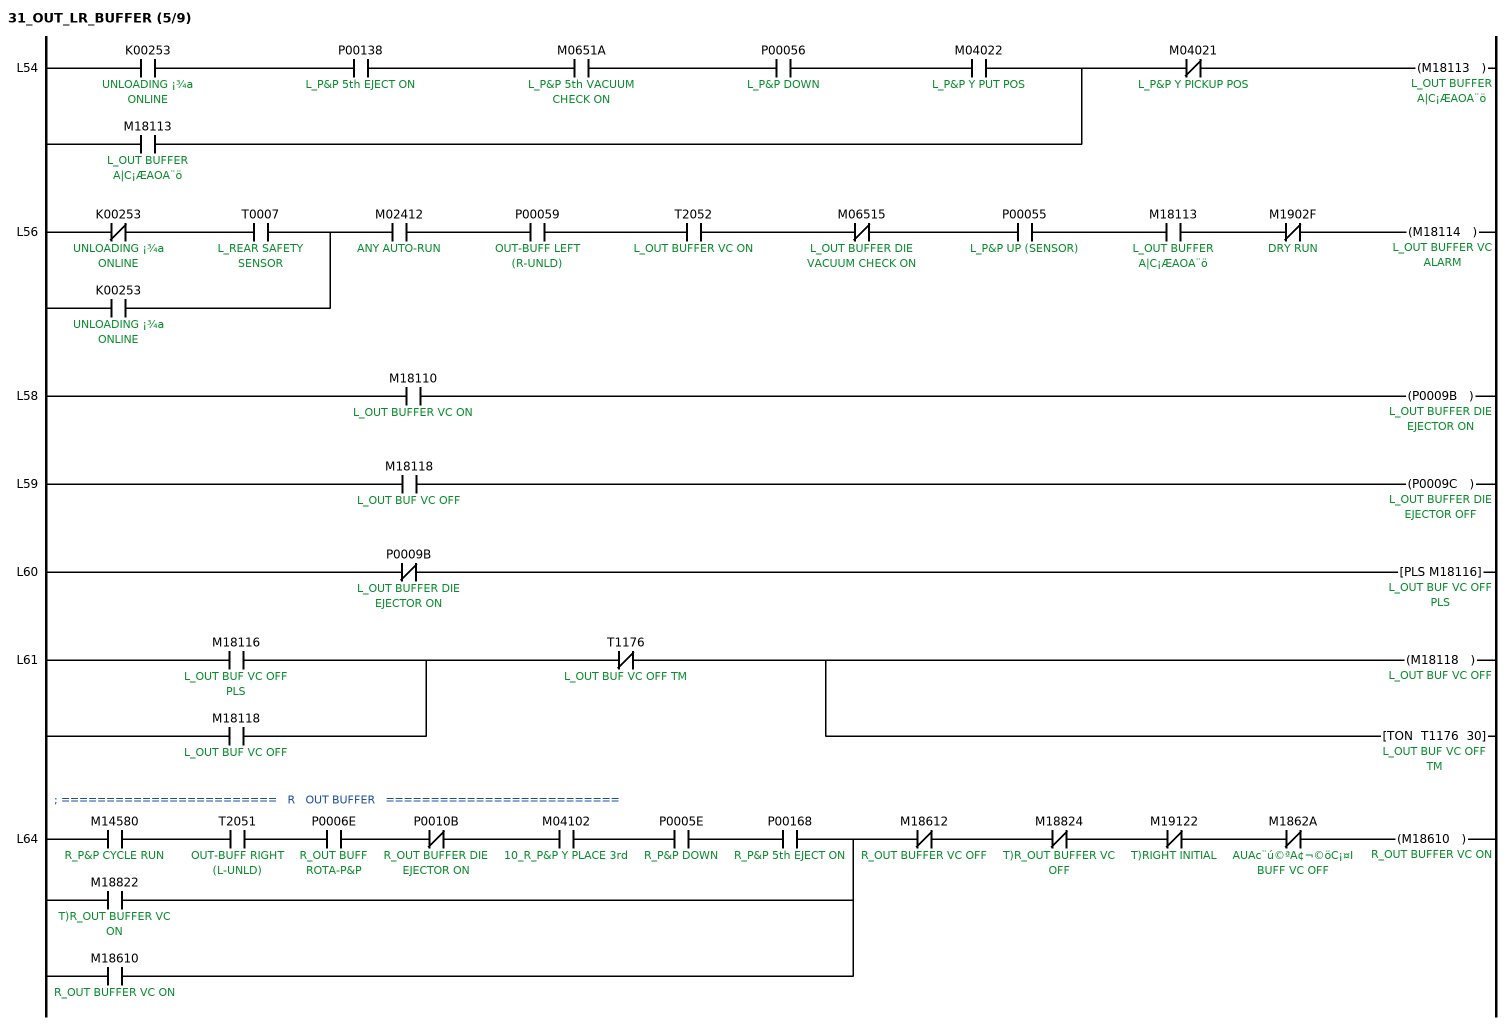
; L54
LOAD      K00253	// UNLOADING ¡¾a ONLINE
AND       P00138	// L_P&P 5th EJECT ON
AND       M0651A	// L_P&P 5th VACUUM CHECK ON
AND       P00056	// L_P&P DOWN
AND       M04022	// L_P&P Y PUT POS
OR        M18113	// L_OUT BUFFER A|C¡ÆAOA¨ö
AND NOT   M04021	// L_P&P Y PICKUP POS
OUT       M18113	// L_OUT BUFFER A|C¡ÆAOA¨ö
; L56
LOAD NOT  K00253	// UNLOADING ¡¾a ONLINE
AND       T0007	// L_REAR SAFETY SENSOR
OR        K00253	// UNLOADING ¡¾a ONLINE
AND       M02412	// ANY AUTO-RUN
AND       P00059	// OUT-BUFF LEFT (R-UNLD)
AND       T2052	// L_OUT BUFFER VC ON
AND NOT   M06515	// L_OUT BUFFER DIE VACUUM CHECK ON
AND       P00055	// L_P&P UP (SENSOR)
AND       M18113	// L_OUT BUFFER A|C¡ÆAOA¨ö
AND NOT   M1902F	// DRY RUN
OUT       M18114	// L_OUT BUFFER VC ALARM
; L58
LOAD      M18110	// L_OUT BUFFER VC ON
OUT       P0009B	// L_OUT BUFFER DIE EJECTOR ON
; L59
LOAD      M18118	// L_OUT BUF VC OFF
OUT       P0009C	// L_OUT BUFFER DIE EJECTOR OFF
; L60
LOAD NOT  P0009B	// L_OUT BUFFER DIE EJECTOR ON
OUTP      M18116	// L_OUT BUF VC OFF PLS
; L61
LOAD      M18116	// L_OUT BUF VC OFF PLS
OR        M18118	// L_OUT BUF VC OFF
AND NOT   T1176	// L_OUT BUF VC OFF TM
OUT       M18118	// L_OUT BUF VC OFF
TON       T1176 30	// L_OUT BUF VC OFF TM
// ========================   R   OUT BUFFER   ==========================
; L64
LOAD      M14580	// R_P&P CYCLE RUN
AND       T2051	// OUT-BUFF RIGHT (L-UNLD)
AND       P0006E	// R_OUT BUFF ROTA-P&P
AND NOT   P0010B	// R_OUT BUFFER DIE EJECTOR ON
AND       M04102	// 10_R_P&P Y PLACE 3rd
AND       P0005E	// R_P&P DOWN
AND       P00168	// R_P&P 5th EJECT ON
OR        M18822	// T)R_OUT BUFFER VC ON
OR        M18610	// R_OUT BUFFER VC ON
AND NOT   M18612	// R_OUT BUFFER VC OFF
AND NOT   M18824	// T)R_OUT BUFFER VC OFF
AND NOT   M19122	// T)RIGHT INITIAL
AND NOT   M1862A	// AUAc¨ú©ªA¢¬©öC¡¤I BUFF VC OFF
OUT       M18610	// R_OUT BUFFER VC ON

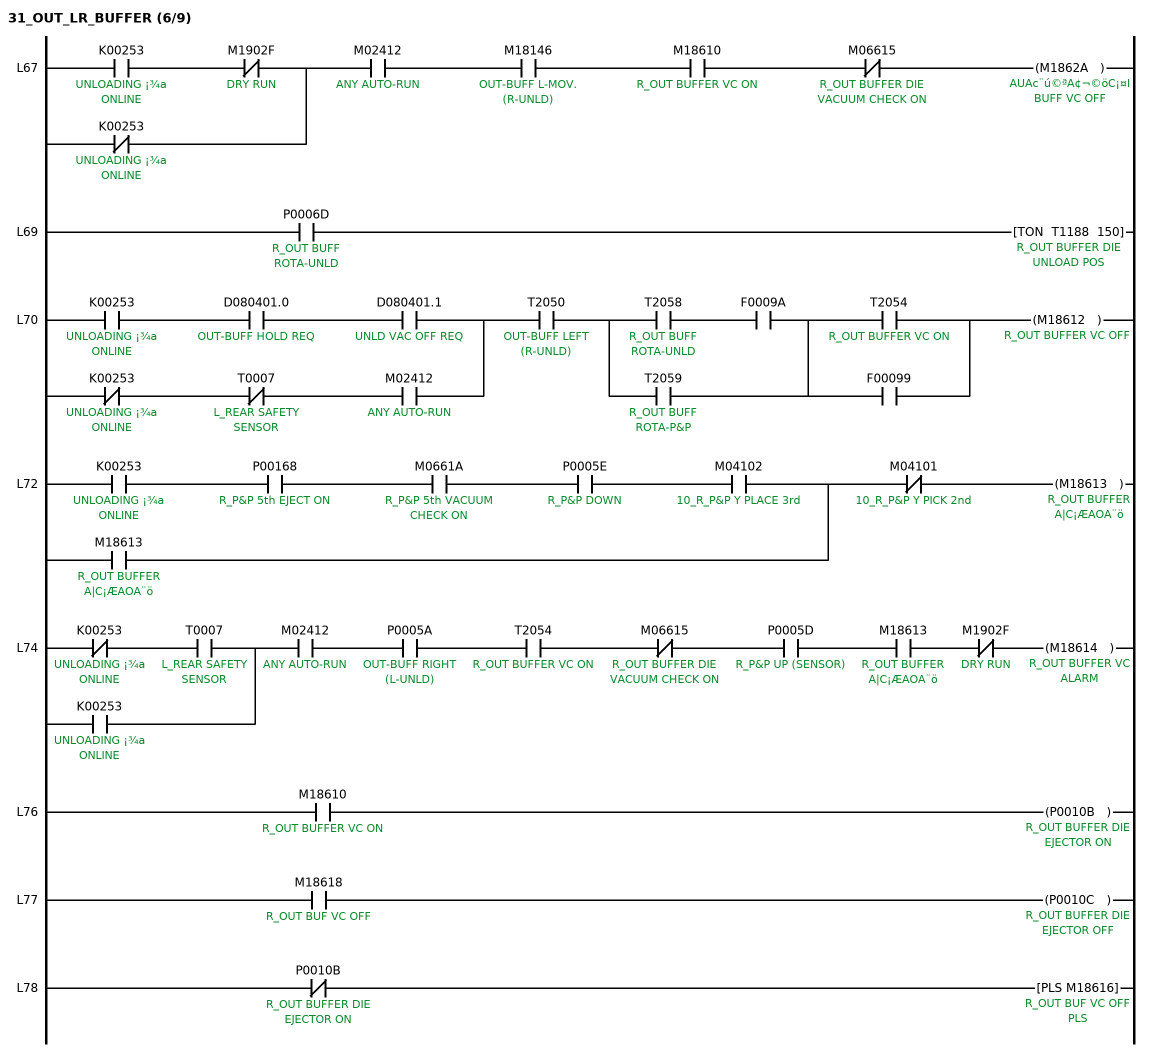
; L67
LOAD      K00253	// UNLOADING ¡¾a ONLINE
AND NOT   M1902F	// DRY RUN
OR NOT    K00253	// UNLOADING ¡¾a ONLINE
AND       M02412	// ANY AUTO-RUN
AND       M18146	// OUT-BUFF L-MOV.  (R-UNLD)
AND       M18610	// R_OUT BUFFER VC ON
AND NOT   M06615	// R_OUT BUFFER DIE VACUUM CHECK ON
OUT       M1862A	// AUAc¨ú©ªA¢¬©öC¡¤I BUFF VC OFF
; L69
LOAD      P0006D	// R_OUT BUFF ROTA-UNLD
TON       T1188 150	// R_OUT BUFFER DIE UNLOAD POS
; L70
LOAD      K00253	// UNLOADING ¡¾a ONLINE
AND       D080401.0	// OUT-BUFF HOLD REQ
AND       D080401.1	// UNLD VAC OFF REQ
LOAD NOT  K00253	// UNLOADING ¡¾a ONLINE
AND NOT   T0007	// L_REAR SAFETY SENSOR
AND       M02412	// ANY AUTO-RUN
OR LOAD
AND       T2050	// OUT-BUFF LEFT (R-UNLD)
LOAD      T2058	// R_OUT BUFF ROTA-UNLD
AND       F0009A
OR        T2059	// R_OUT BUFF ROTA-P&P
AND LOAD
LOAD      T2054	// R_OUT BUFFER VC ON
OR        F00099
AND LOAD
OUT       M18612	// R_OUT BUFFER VC OFF
; L72
LOAD      K00253	// UNLOADING ¡¾a ONLINE
AND       P00168	// R_P&P 5th EJECT ON
AND       M0661A	// R_P&P 5th VACUUM CHECK ON
AND       P0005E	// R_P&P DOWN
AND       M04102	// 10_R_P&P Y PLACE 3rd
OR        M18613	// R_OUT BUFFER A|C¡ÆAOA¨ö
AND NOT   M04101	// 10_R_P&P Y PICK 2nd
OUT       M18613	// R_OUT BUFFER A|C¡ÆAOA¨ö
; L74
LOAD NOT  K00253	// UNLOADING ¡¾a ONLINE
AND       T0007	// L_REAR SAFETY SENSOR
OR        K00253	// UNLOADING ¡¾a ONLINE
AND       M02412	// ANY AUTO-RUN
AND       P0005A	// OUT-BUFF RIGHT (L-UNLD)
AND       T2054	// R_OUT BUFFER VC ON
AND NOT   M06615	// R_OUT BUFFER DIE VACUUM CHECK ON
AND       P0005D	// R_P&P UP (SENSOR)
AND       M18613	// R_OUT BUFFER A|C¡ÆAOA¨ö
AND NOT   M1902F	// DRY RUN
OUT       M18614	// R_OUT BUFFER VC ALARM
; L76
LOAD      M18610	// R_OUT BUFFER VC ON
OUT       P0010B	// R_OUT BUFFER DIE EJECTOR ON
; L77
LOAD      M18618	// R_OUT BUF VC OFF
OUT       P0010C	// R_OUT BUFFER DIE EJECTOR OFF
; L78
LOAD NOT  P0010B	// R_OUT BUFFER DIE EJECTOR ON
OUTP      M18616	// R_OUT BUF VC OFF PLS

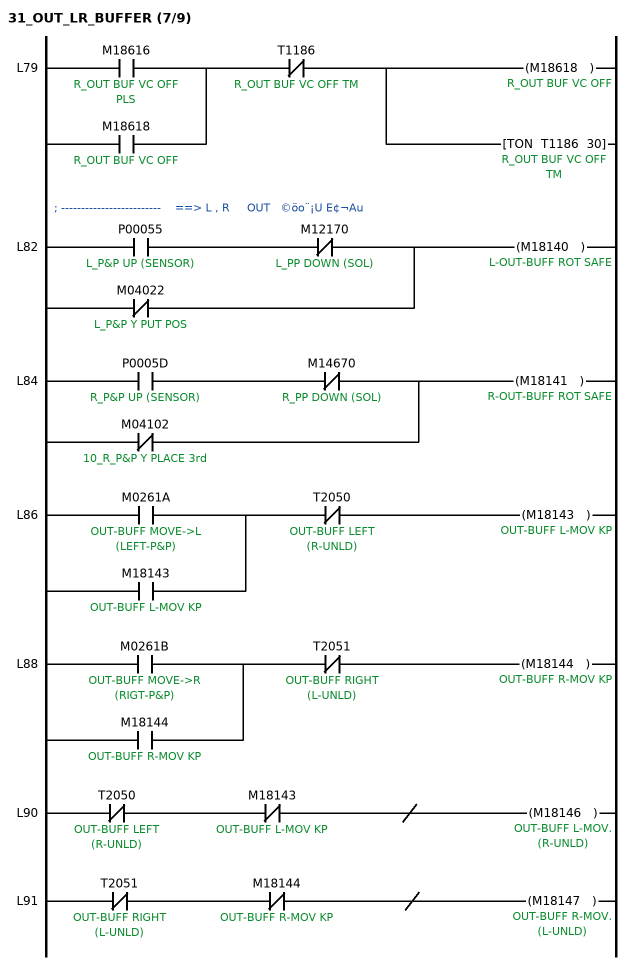
; L79
LOAD      M18616	// R_OUT BUF VC OFF PLS
OR        M18618	// R_OUT BUF VC OFF
AND NOT   T1186	// R_OUT BUF VC OFF TM
OUT       M18618	// R_OUT BUF VC OFF
TON       T1186 30	// R_OUT BUF VC OFF TM
// -------------------------    ==> L , R     OUT   ©öo¨¡U E¢¬Au
; L82
LOAD      P00055	// L_P&P UP (SENSOR)
AND NOT   M12170	// L_PP DOWN (SOL)
OR NOT    M04022	// L_P&P Y PUT POS
OUT       M18140	// L-OUT-BUFF ROT SAFE
; L84
LOAD      P0005D	// R_P&P UP (SENSOR)
AND NOT   M14670	// R_PP DOWN (SOL)
OR NOT    M04102	// 10_R_P&P Y PLACE 3rd
OUT       M18141	// R-OUT-BUFF ROT SAFE
; L86
LOAD      M0261A	// OUT-BUFF MOVE->L (LEFT-P&P)
OR        M18143	// OUT-BUFF L-MOV KP
AND NOT   T2050	// OUT-BUFF LEFT (R-UNLD)
OUT       M18143	// OUT-BUFF L-MOV KP
; L88
LOAD      M0261B	// OUT-BUFF MOVE->R (RIGT-P&P)
OR        M18144	// OUT-BUFF R-MOV KP
AND NOT   T2051	// OUT-BUFF RIGHT (L-UNLD)
OUT       M18144	// OUT-BUFF R-MOV KP
; L90
LOAD NOT  T2050	// OUT-BUFF LEFT (R-UNLD)
AND NOT   M18143	// OUT-BUFF L-MOV KP
NOT
OUT       M18146	// OUT-BUFF L-MOV.  (R-UNLD)
; L91
LOAD NOT  T2051	// OUT-BUFF RIGHT (L-UNLD)
AND NOT   M18144	// OUT-BUFF R-MOV KP
NOT
OUT       M18147	// OUT-BUFF R-MOV.  (L-UNLD)

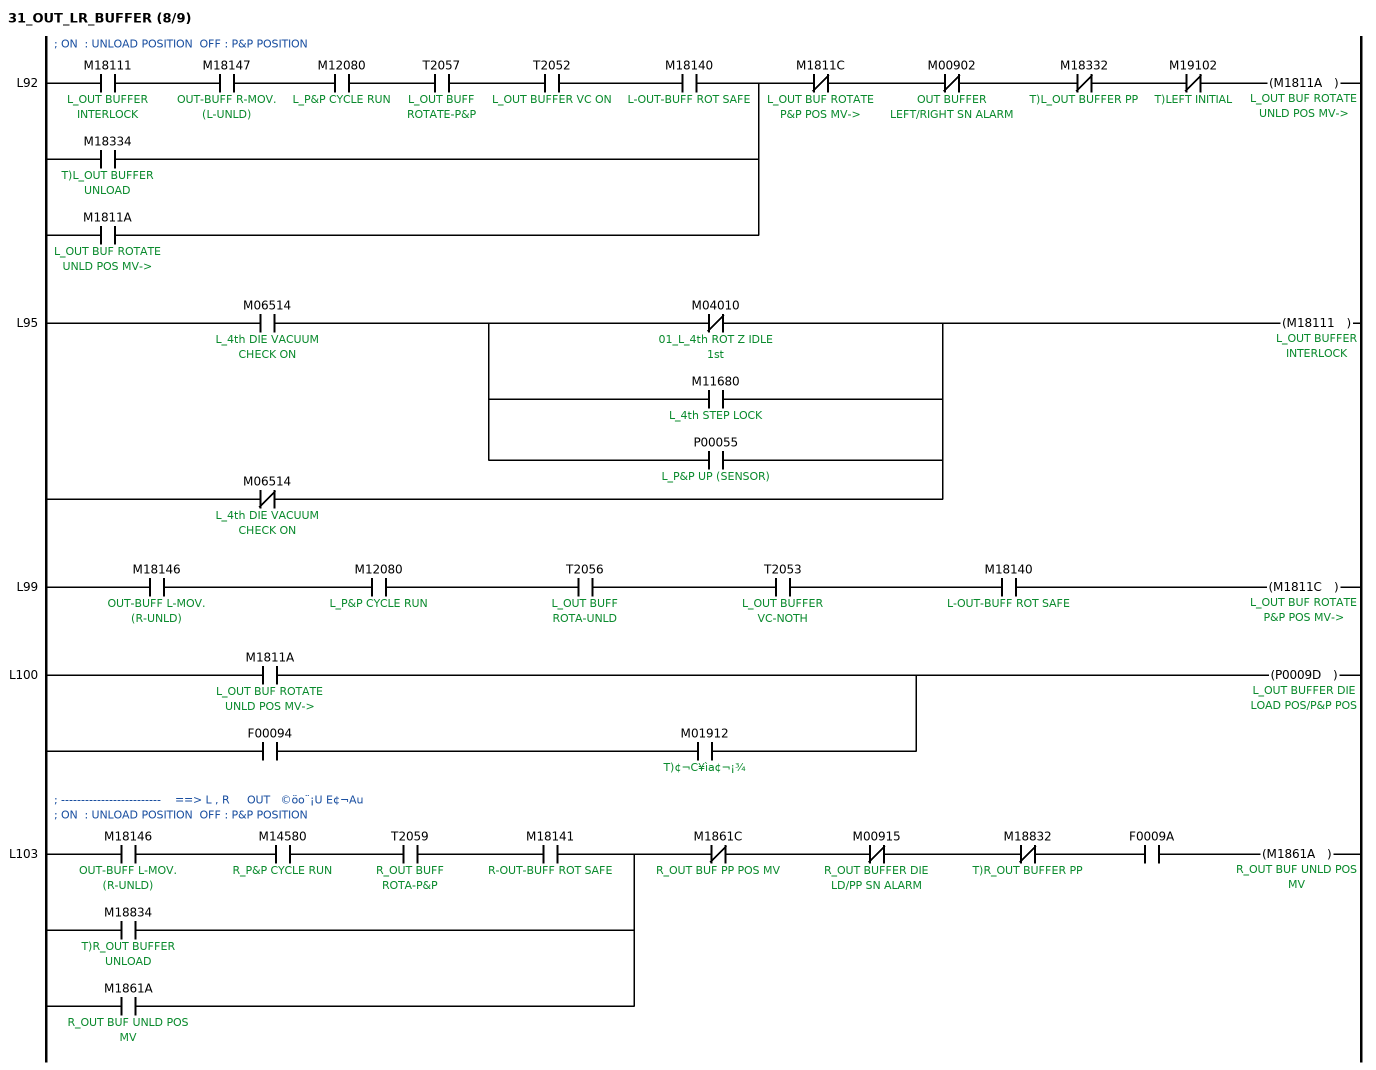
; L92
LOAD      M18111	// L_OUT BUFFER INTERLOCK
AND       M18147	// OUT-BUFF R-MOV.  (L-UNLD)
AND       M12080	// L_P&P CYCLE RUN
AND       T2057	// L_OUT BUFF ROTATE-P&P
AND       T2052	// L_OUT BUFFER VC ON
AND       M18140	// L-OUT-BUFF ROT SAFE
OR        M18334	// T)L_OUT BUFFER UNLOAD
OR        M1811A	// L_OUT BUF ROTATE UNLD POS MV->
AND NOT   M1811C	// L_OUT BUF ROTATE P&P POS MV->
AND NOT   M00902	// OUT BUFFER LEFT/RIGHT SN ALARM
AND NOT   M18332	// T)L_OUT BUFFER PP
AND NOT   M19102	// T)LEFT INITIAL
OUT       M1811A	// L_OUT BUF ROTATE UNLD POS MV->
// output comment: ON  : UNLOAD POSITION  OFF : P&P POSITION
; L95
LOAD      M06514	// L_4th DIE VACUUM CHECK ON
LOAD NOT  M04010	// 01_L_4th ROT Z IDLE 1st
OR        M11680	// L_4th STEP LOCK
OR        P00055	// L_P&P UP (SENSOR)
AND LOAD
OR NOT    M06514	// L_4th DIE VACUUM CHECK ON
OUT       M18111	// L_OUT BUFFER INTERLOCK
; L99
LOAD      M18146	// OUT-BUFF L-MOV.  (R-UNLD)
AND       M12080	// L_P&P CYCLE RUN
AND       T2056	// L_OUT BUFF ROTA-UNLD
AND       T2053	// L_OUT BUFFER VC-NOTH
AND       M18140	// L-OUT-BUFF ROT SAFE
OUT       M1811C	// L_OUT BUF ROTATE P&P POS MV->
; L100
LOAD      M1811A	// L_OUT BUF ROTATE UNLD POS MV->
LOAD      F00094
AND       M01912	// T)¢¬C¥ìa¢¬¡¾
OR LOAD
OUT       P0009D	// L_OUT BUFFER DIE LOAD POS/P&P POS
// -------------------------    ==> L , R     OUT   ©öo¨¡U E¢¬Au
; L103
LOAD      M18146	// OUT-BUFF L-MOV.  (R-UNLD)
AND       M14580	// R_P&P CYCLE RUN
AND       T2059	// R_OUT BUFF ROTA-P&P
AND       M18141	// R-OUT-BUFF ROT SAFE
OR        M18834	// T)R_OUT BUFFER UNLOAD
OR        M1861A	// R_OUT BUF UNLD POS MV
AND NOT   M1861C	// R_OUT BUF PP POS MV
AND NOT   M00915	// R_OUT BUFFER DIE LD/PP SN ALARM
AND NOT   M18832	// T)R_OUT BUFFER PP
AND       F0009A
OUT       M1861A	// R_OUT BUF UNLD POS MV
// output comment: ON  : UNLOAD POSITION  OFF : P&P POSITION

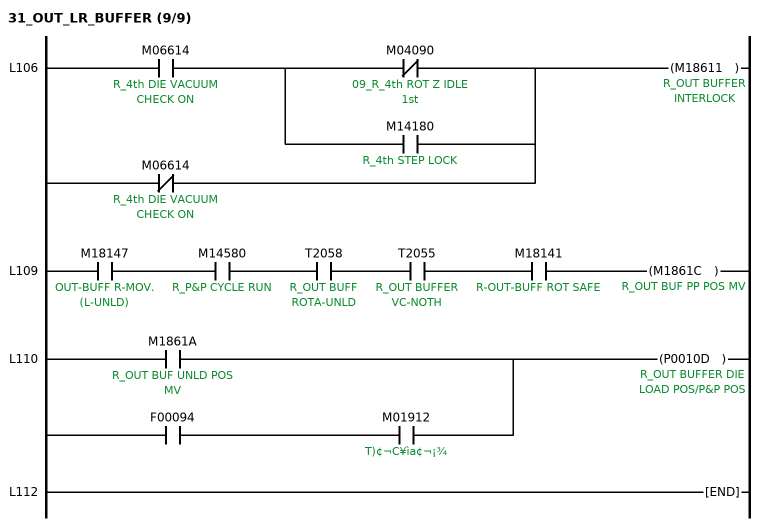
; L106
LOAD      M06614	// R_4th DIE VACUUM CHECK ON
LOAD NOT  M04090	// 09_R_4th ROT Z IDLE 1st
OR        M14180	// R_4th STEP LOCK
AND LOAD
OR NOT    M06614	// R_4th DIE VACUUM CHECK ON
OUT       M18611	// R_OUT BUFFER INTERLOCK
; L109
LOAD      M18147	// OUT-BUFF R-MOV.  (L-UNLD)
AND       M14580	// R_P&P CYCLE RUN
AND       T2058	// R_OUT BUFF ROTA-UNLD
AND       T2055	// R_OUT BUFFER VC-NOTH
AND       M18141	// R-OUT-BUFF ROT SAFE
OUT       M1861C	// R_OUT BUF PP POS MV
; L110
LOAD      M1861A	// R_OUT BUF UNLD POS MV
LOAD      F00094
AND       M01912	// T)¢¬C¥ìa¢¬¡¾
OR LOAD
OUT       P0010D	// R_OUT BUFFER DIE LOAD POS/P&P POS
; L112
END

PROGRAM 40_2D_CODE (task: ¨ö¨¬A¥ì CA¡¤I¡¾¡¿¡¤¡Í)

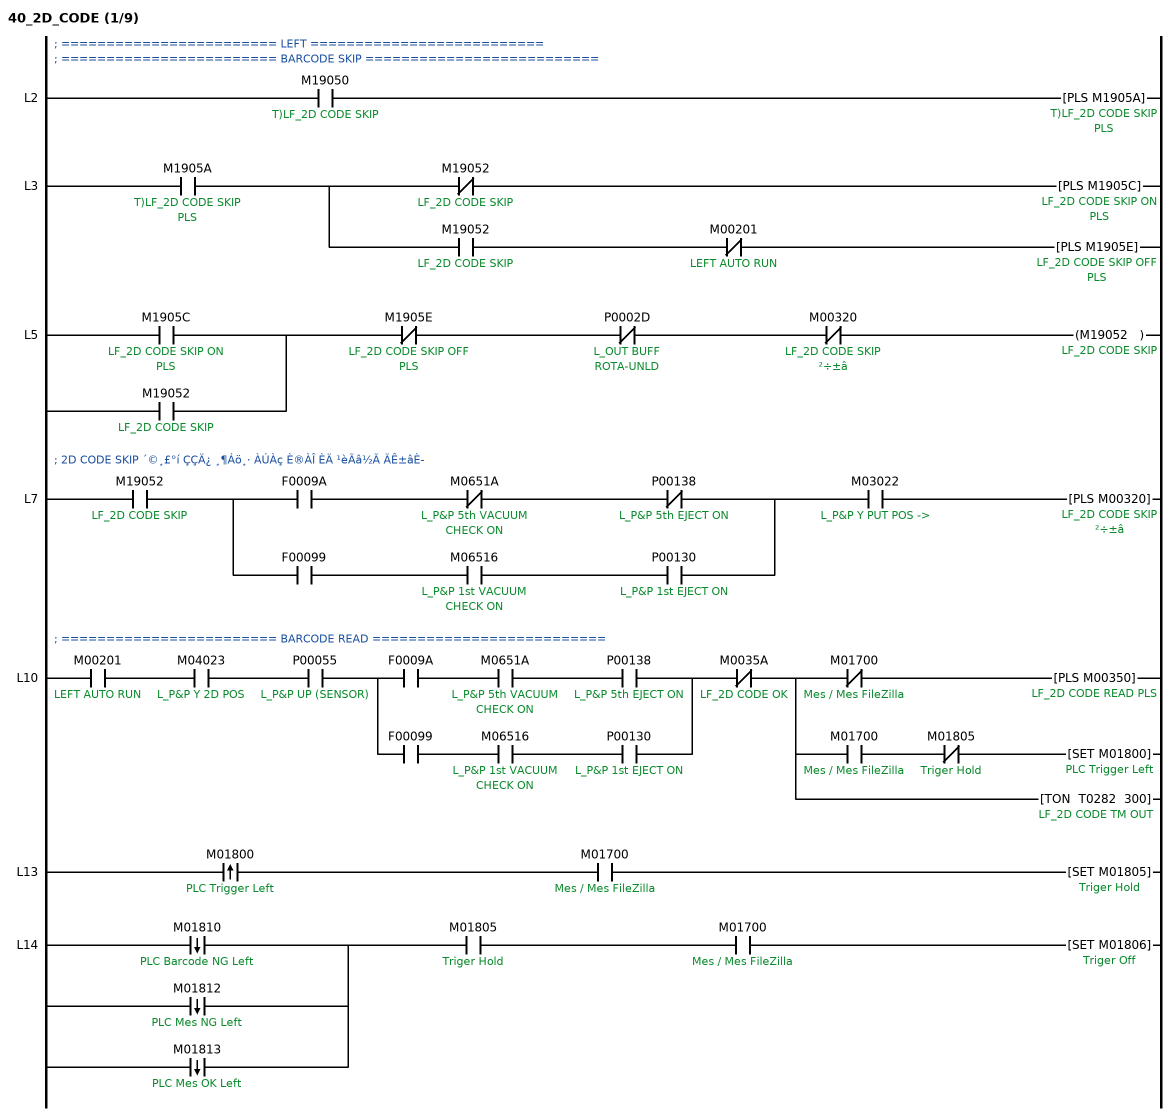
// ======================== LEFT ==========================
// ======================== BARCODE SKIP ==========================
; L2
LOAD      M19050	// T)LF_2D CODE SKIP
OUTP      M1905A	// T)LF_2D CODE SKIP PLS
; L3
LOAD      M1905A	// T)LF_2D CODE SKIP PLS
MPUSH
AND NOT   M19052	// LF_2D CODE SKIP
OUTP      M1905C	// LF_2D CODE SKIP ON PLS
MPOP
AND       M19052	// LF_2D CODE SKIP
AND NOT   M00201	// LEFT AUTO RUN
OUTP      M1905E	// LF_2D CODE SKIP OFF PLS
; L5
LOAD      M1905C	// LF_2D CODE SKIP ON PLS
OR        M19052	// LF_2D CODE SKIP
AND NOT   M1905E	// LF_2D CODE SKIP OFF PLS
AND NOT   P0002D	// L_OUT BUFF ROTA-UNLD
AND NOT   M00320	// LF_2D CODE SKIP ²÷±â
OUT       M19052	// LF_2D CODE SKIP
; L7
LOAD      M19052	// LF_2D CODE SKIP
LOAD      F0009A
AND NOT   M0651A	// L_P&P 5th VACUUM CHECK ON
AND NOT   P00138	// L_P&P 5th EJECT ON
LOAD      F00099
AND       M06516	// L_P&P 1st VACUUM CHECK ON
AND       P00130	// L_P&P 1st EJECT ON
OR LOAD
AND LOAD
AND       M03022	// L_P&P Y PUT POS ->
OUTP      M00320	// LF_2D CODE SKIP ²÷±â
// output comment: 2D CODE SKIP ´©¸£°í ÇÇÄ¿ ¸¶Áö¸· ÀÚÀç È®ÀÎ ÈÄ ¹èÃâ½Ã ÃÊ±âÈ­
// ======================== BARCODE READ ==========================
; L10
LOAD      M00201	// LEFT AUTO RUN
AND       M04023	// L_P&P Y 2D POS
AND       P00055	// L_P&P UP (SENSOR)
LOAD      F0009A
AND       M0651A	// L_P&P 5th VACUUM CHECK ON
AND       P00138	// L_P&P 5th EJECT ON
LOAD      F00099
AND       M06516	// L_P&P 1st VACUUM CHECK ON
AND       P00130	// L_P&P 1st EJECT ON
OR LOAD
AND LOAD
AND NOT   M0035A	// LF_2D CODE OK
MPUSH
AND NOT   M01700	// Mes / Mes FileZilla
OUTP      M00350	// LF_2D CODE READ PLS
MLOAD
AND       M01700	// Mes / Mes FileZilla
AND NOT   M01805	// Triger Hold
SET       M01800	// PLC Trigger Left
MPOP
TON       T0282 300	// LF_2D CODE TM OUT
; L13
LOADP     M01800	// PLC Trigger Left
AND       M01700	// Mes / Mes FileZilla
SET       M01805	// Triger Hold
; L14
LOADN     M01810	// PLC Barcode NG Left
ORN       M01812	// PLC Mes NG Left
ORN       M01813	// PLC Mes OK Left
AND       M01805	// Triger Hold
AND       M01700	// Mes / Mes FileZilla
SET       M01806	// Triger Off

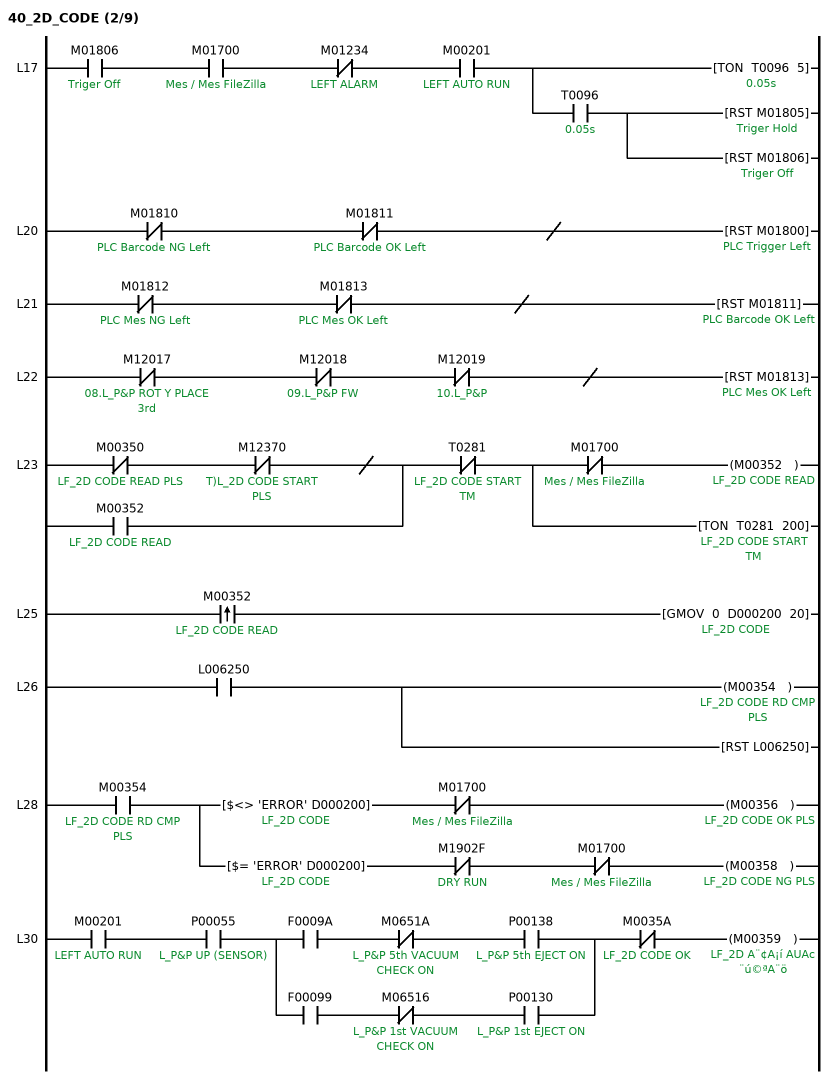
; L17
LOAD      M01806	// Triger Off
AND       M01700	// Mes / Mes FileZilla
AND NOT   M01234	// LEFT ALARM
AND       M00201	// LEFT AUTO RUN
TON       T0096 5	// 0.05s
AND       T0096	// 0.05s
RST       M01805	// Triger Hold
RST       M01806	// Triger Off
; L20
LOAD NOT  M01810	// PLC Barcode NG Left
AND NOT   M01811	// PLC Barcode OK Left
NOT
RST       M01800	// PLC Trigger Left
; L21
LOAD NOT  M01812	// PLC Mes NG Left
AND NOT   M01813	// PLC Mes OK Left
NOT
RST       M01811	// PLC Barcode OK Left
; L22
LOAD NOT  M12017	// 08.L_P&P ROT Y PLACE 3rd
AND NOT   M12018	// 09.L_P&P FW
AND NOT   M12019	// 10.L_P&P
NOT
RST       M01813	// PLC Mes OK Left
; L23
LOAD NOT  M00350	// LF_2D CODE READ PLS
AND NOT   M12370	// T)L_2D CODE START PLS
NOT
OR        M00352	// LF_2D CODE READ
AND NOT   T0281	// LF_2D CODE START TM
MPUSH
AND NOT   M01700	// Mes / Mes FileZilla
OUT       M00352	// LF_2D CODE READ
MPOP
TON       T0281 200	// LF_2D CODE START TM
; L25
LOADP     M00352	// LF_2D CODE READ
GMOV      0 D000200 20	// LF_2D CODE
; L26
LOAD      L006250
OUT       M00354	// LF_2D CODE RD CMP PLS
RST       L006250
; L28
LOAD      M00354	// LF_2D CODE RD CMP PLS
MPUSH
AND$<>    'ERROR' D000200	// LF_2D CODE
AND NOT   M01700	// Mes / Mes FileZilla
OUT       M00356	// LF_2D CODE OK PLS
MPOP
AND$=     'ERROR' D000200	// LF_2D CODE
AND NOT   M1902F	// DRY RUN
AND NOT   M01700	// Mes / Mes FileZilla
OUT       M00358	// LF_2D CODE NG PLS
; L30
LOAD      M00201	// LEFT AUTO RUN
AND       P00055	// L_P&P UP (SENSOR)
LOAD      F0009A
AND NOT   M0651A	// L_P&P 5th VACUUM CHECK ON
AND       P00138	// L_P&P 5th EJECT ON
LOAD      F00099
AND NOT   M06516	// L_P&P 1st VACUUM CHECK ON
AND       P00130	// L_P&P 1st EJECT ON
OR LOAD
AND LOAD
AND NOT   M0035A	// LF_2D CODE OK
OUT       M00359	// LF_2D A¨¢A¡í AUAc ¨ú©ªA¨ö

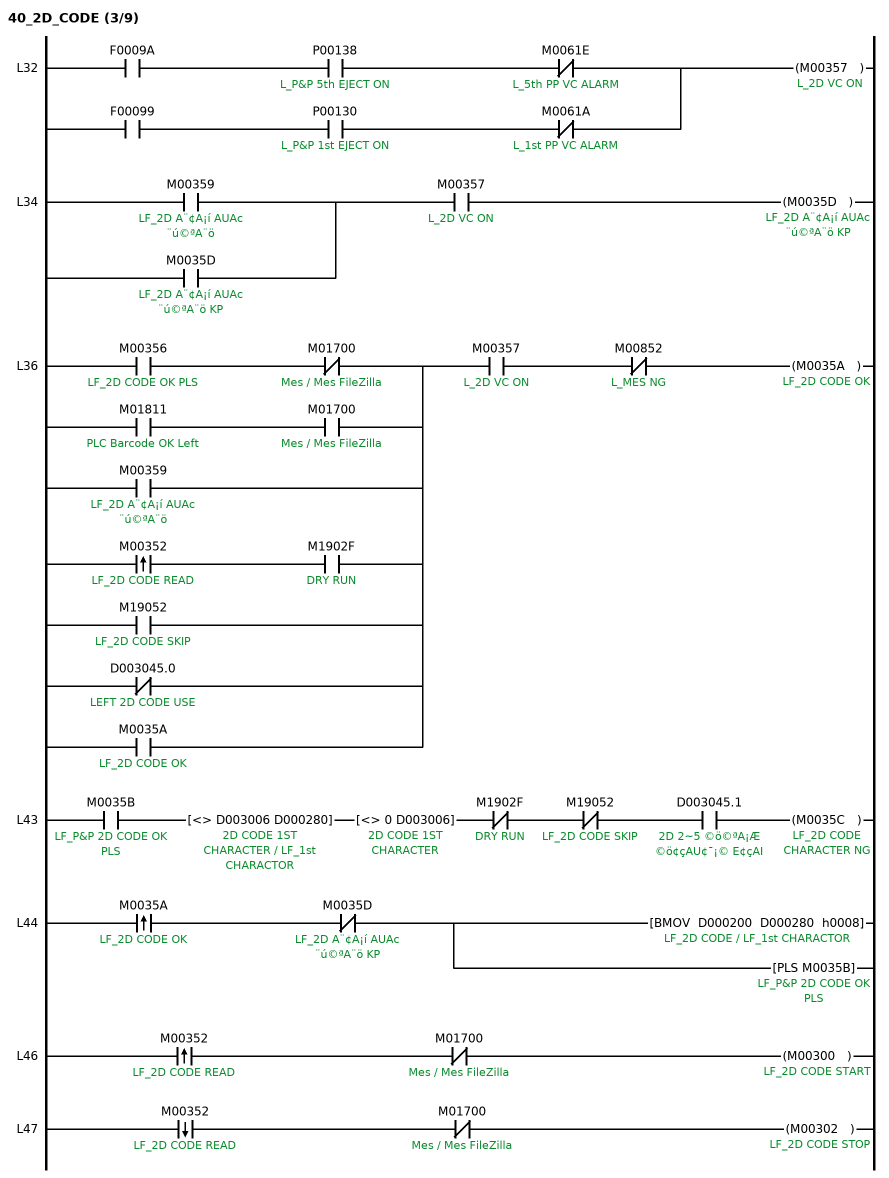
; L32
LOAD      F0009A
AND       P00138	// L_P&P 5th EJECT ON
AND NOT   M0061E	// L_5th PP VC ALARM
LOAD      F00099
AND       P00130	// L_P&P 1st EJECT ON
AND NOT   M0061A	// L_1st PP VC ALARM
OR LOAD
OUT       M00357	// L_2D VC ON
; L34
LOAD      M00359	// LF_2D A¨¢A¡í AUAc ¨ú©ªA¨ö
OR        M0035D	// LF_2D A¨¢A¡í AUAc ¨ú©ªA¨ö KP
AND       M00357	// L_2D VC ON
OUT       M0035D	// LF_2D A¨¢A¡í AUAc ¨ú©ªA¨ö KP
; L36
LOAD      M00356	// LF_2D CODE OK PLS
AND NOT   M01700	// Mes / Mes FileZilla
LOAD      M01811	// PLC Barcode OK Left
AND       M01700	// Mes / Mes FileZilla
OR LOAD
OR        M00359	// LF_2D A¨¢A¡í AUAc ¨ú©ªA¨ö
LOADP     M00352	// LF_2D CODE READ
AND       M1902F	// DRY RUN
OR LOAD
OR        M19052	// LF_2D CODE SKIP
OR NOT    D003045.0	// LEFT 2D CODE USE
OR        M0035A	// LF_2D CODE OK
AND       M00357	// L_2D VC ON
AND NOT   M00852	// L_MES NG
OUT       M0035A	// LF_2D CODE OK
; L43
LOAD      M0035B	// LF_P&P 2D CODE OK PLS
AND<>     D003006 D000280	// 2D CODE 1ST CHARACTER / LF_1st CHARACTOR
AND<>     0 D003006	// 2D CODE 1ST CHARACTER
AND NOT   M1902F	// DRY RUN
AND NOT   M19052	// LF_2D CODE SKIP
AND       D003045.1	// 2D 2~5 ©ö©ªA¡Æ ©ö¢çAU¢¯¡© E¢çAI
OUT       M0035C	// LF_2D CODE CHARACTER NG
; L44
LOADP     M0035A	// LF_2D CODE OK
AND NOT   M0035D	// LF_2D A¨¢A¡í AUAc ¨ú©ªA¨ö KP
BMOV      D000200 D000280 h0008	// LF_2D CODE / LF_1st CHARACTOR
OUTP      M0035B	// LF_P&P 2D CODE OK PLS
; L46
LOADP     M00352	// LF_2D CODE READ
AND NOT   M01700	// Mes / Mes FileZilla
OUT       M00300	// LF_2D CODE START
; L47
LOADN     M00352	// LF_2D CODE READ
AND NOT   M01700	// Mes / Mes FileZilla
OUT       M00302	// LF_2D CODE STOP

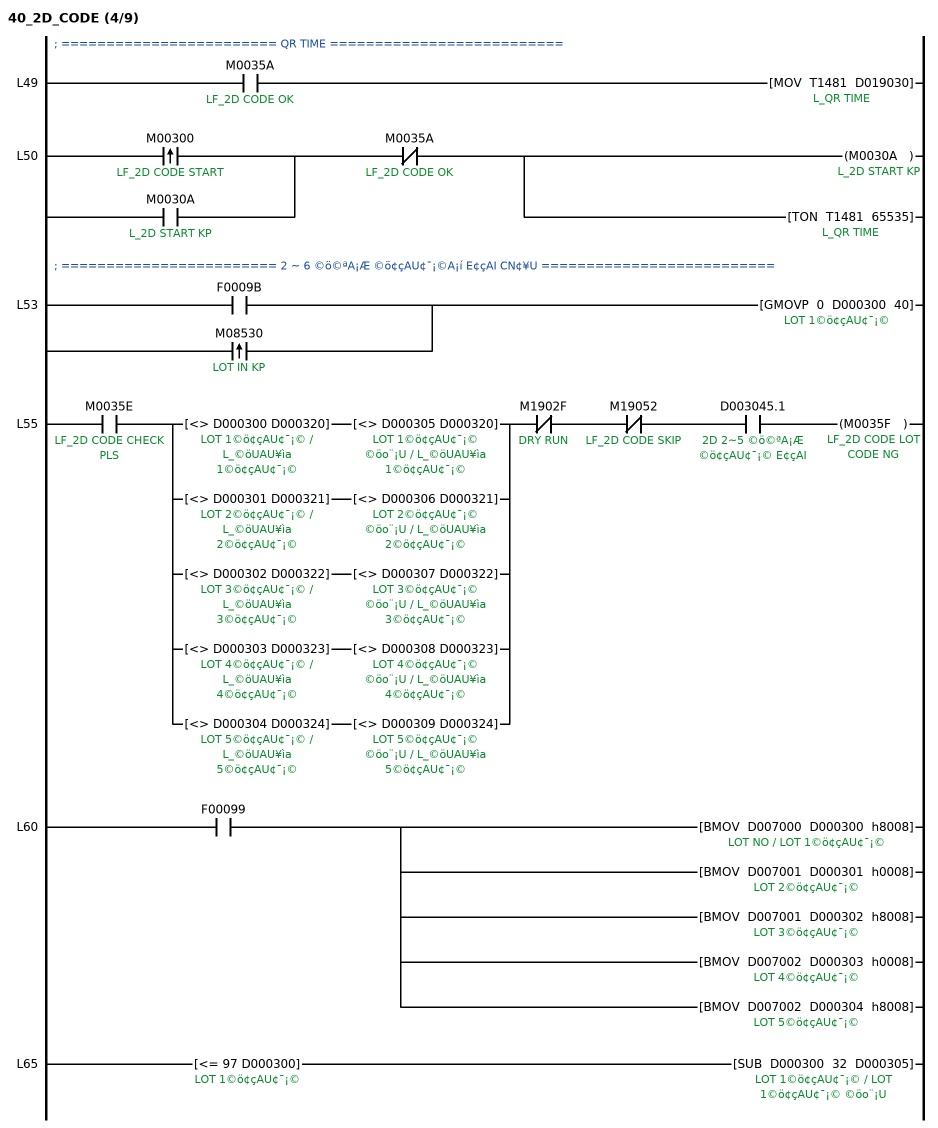
// ======================== QR TIME ==========================
; L49
LOAD      M0035A	// LF_2D CODE OK
MOV       T1481 D019030	// L_QR TIME
; L50
LOADP     M00300	// LF_2D CODE START
OR        M0030A	// L_2D START KP
AND NOT   M0035A	// LF_2D CODE OK
OUT       M0030A	// L_2D START KP
TON       T1481 65535	// L_QR TIME
// ======================== 2 ~ 6 ©ö©ªA¡Æ ©ö¢çAU¢¯¡©A¡í E¢çAI CN¢¥U ==========================
; L53
LOAD      F0009B
ORP       M08530	// LOT IN KP
GMOVP     0 D000300 40	// LOT 1©ö¢çAU¢¯¡©
; L55
LOAD      M0035E	// LF_2D CODE CHECK PLS
LOAD<>    D000300 D000320	// LOT 1©ö¢çAU¢¯¡© / L_©öUAU¥ìa 1©ö¢çAU¢¯¡©
AND<>     D000305 D000320	// LOT 1©ö¢çAU¢¯¡© ©öo¨¡U / L_©öUAU¥ìa 1©ö¢çAU¢¯¡©
LOAD<>    D000301 D000321	// LOT 2©ö¢çAU¢¯¡© / L_©öUAU¥ìa 2©ö¢çAU¢¯¡©
AND<>     D000306 D000321	// LOT 2©ö¢çAU¢¯¡© ©öo¨¡U / L_©öUAU¥ìa 2©ö¢çAU¢¯¡©
OR LOAD
LOAD<>    D000302 D000322	// LOT 3©ö¢çAU¢¯¡© / L_©öUAU¥ìa 3©ö¢çAU¢¯¡©
AND<>     D000307 D000322	// LOT 3©ö¢çAU¢¯¡© ©öo¨¡U / L_©öUAU¥ìa 3©ö¢çAU¢¯¡©
OR LOAD
LOAD<>    D000303 D000323	// LOT 4©ö¢çAU¢¯¡© / L_©öUAU¥ìa 4©ö¢çAU¢¯¡©
AND<>     D000308 D000323	// LOT 4©ö¢çAU¢¯¡© ©öo¨¡U / L_©öUAU¥ìa 4©ö¢çAU¢¯¡©
OR LOAD
LOAD<>    D000304 D000324	// LOT 5©ö¢çAU¢¯¡© / L_©öUAU¥ìa 5©ö¢çAU¢¯¡©
AND<>     D000309 D000324	// LOT 5©ö¢çAU¢¯¡© ©öo¨¡U / L_©öUAU¥ìa 5©ö¢çAU¢¯¡©
OR LOAD
AND LOAD
AND NOT   M1902F	// DRY RUN
AND NOT   M19052	// LF_2D CODE SKIP
AND       D003045.1	// 2D 2~5 ©ö©ªA¡Æ ©ö¢çAU¢¯¡© E¢çAI
OUT       M0035F	// LF_2D CODE LOT CODE NG
; L60
LOAD      F00099
BMOV      D007000 D000300 h8008	// LOT NO / LOT 1©ö¢çAU¢¯¡©
BMOV      D007001 D000301 h0008	// LOT 2©ö¢çAU¢¯¡©
BMOV      D007001 D000302 h8008	// LOT 3©ö¢çAU¢¯¡©
BMOV      D007002 D000303 h0008	// LOT 4©ö¢çAU¢¯¡©
BMOV      D007002 D000304 h8008	// LOT 5©ö¢çAU¢¯¡©
; L65
LOAD<=    97 D000300	// LOT 1©ö¢çAU¢¯¡©
SUB       D000300 32 D000305	// LOT 1©ö¢çAU¢¯¡© / LOT 1©ö¢çAU¢¯¡© ©öo¨¡U

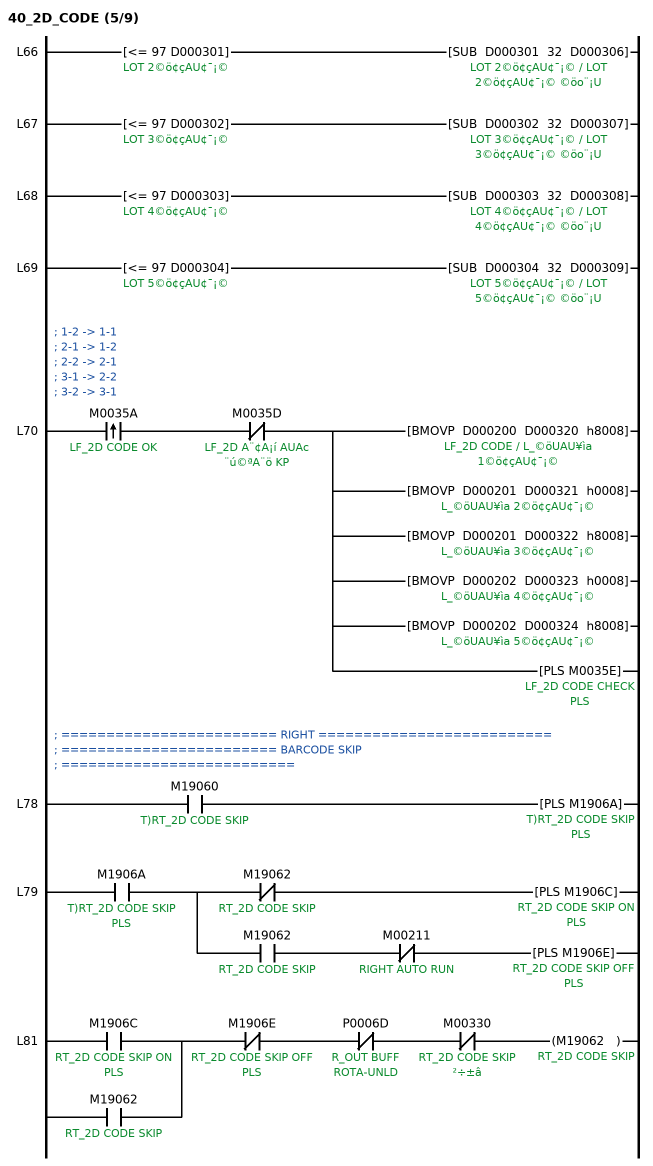
; L66
LOAD<=    97 D000301	// LOT 2©ö¢çAU¢¯¡©
SUB       D000301 32 D000306	// LOT 2©ö¢çAU¢¯¡© / LOT 2©ö¢çAU¢¯¡© ©öo¨¡U
; L67
LOAD<=    97 D000302	// LOT 3©ö¢çAU¢¯¡©
SUB       D000302 32 D000307	// LOT 3©ö¢çAU¢¯¡© / LOT 3©ö¢çAU¢¯¡© ©öo¨¡U
; L68
LOAD<=    97 D000303	// LOT 4©ö¢çAU¢¯¡©
SUB       D000303 32 D000308	// LOT 4©ö¢çAU¢¯¡© / LOT 4©ö¢çAU¢¯¡© ©öo¨¡U
; L69
LOAD<=    97 D000304	// LOT 5©ö¢çAU¢¯¡©
SUB       D000304 32 D000309	// LOT 5©ö¢çAU¢¯¡© / LOT 5©ö¢çAU¢¯¡© ©öo¨¡U
; L70
LOADP     M0035A	// LF_2D CODE OK
AND NOT   M0035D	// LF_2D A¨¢A¡í AUAc ¨ú©ªA¨ö KP
BMOVP     D000200 D000320 h8008	// LF_2D CODE / L_©öUAU¥ìa 1©ö¢çAU¢¯¡©
BMOVP     D000201 D000321 h0008	// L_©öUAU¥ìa 2©ö¢çAU¢¯¡©
BMOVP     D000201 D000322 h8008	// L_©öUAU¥ìa 3©ö¢çAU¢¯¡©
BMOVP     D000202 D000323 h0008	// L_©öUAU¥ìa 4©ö¢çAU¢¯¡©
BMOVP     D000202 D000324 h8008	// L_©öUAU¥ìa 5©ö¢çAU¢¯¡©
OUTP      M0035E	// LF_2D CODE CHECK PLS
// output comment: 1-2 -> 1-1
// output comment: 2-1 -> 1-2
// output comment: 2-2 -> 2-1
// output comment: 3-1 -> 2-2
// output comment: 3-2 -> 3-1
// ======================== RIGHT ==========================
// ======================== BARCODE SKIP ==========================
; L78
LOAD      M19060	// T)RT_2D CODE SKIP
OUTP      M1906A	// T)RT_2D CODE SKIP PLS
; L79
LOAD      M1906A	// T)RT_2D CODE SKIP PLS
MPUSH
AND NOT   M19062	// RT_2D CODE SKIP
OUTP      M1906C	// RT_2D CODE SKIP ON PLS
MPOP
AND       M19062	// RT_2D CODE SKIP
AND NOT   M00211	// RIGHT AUTO RUN
OUTP      M1906E	// RT_2D CODE SKIP OFF PLS
; L81
LOAD      M1906C	// RT_2D CODE SKIP ON PLS
OR        M19062	// RT_2D CODE SKIP
AND NOT   M1906E	// RT_2D CODE SKIP OFF PLS
AND NOT   P0006D	// R_OUT BUFF ROTA-UNLD
AND NOT   M00330	// RT_2D CODE SKIP ²÷±â
OUT       M19062	// RT_2D CODE SKIP

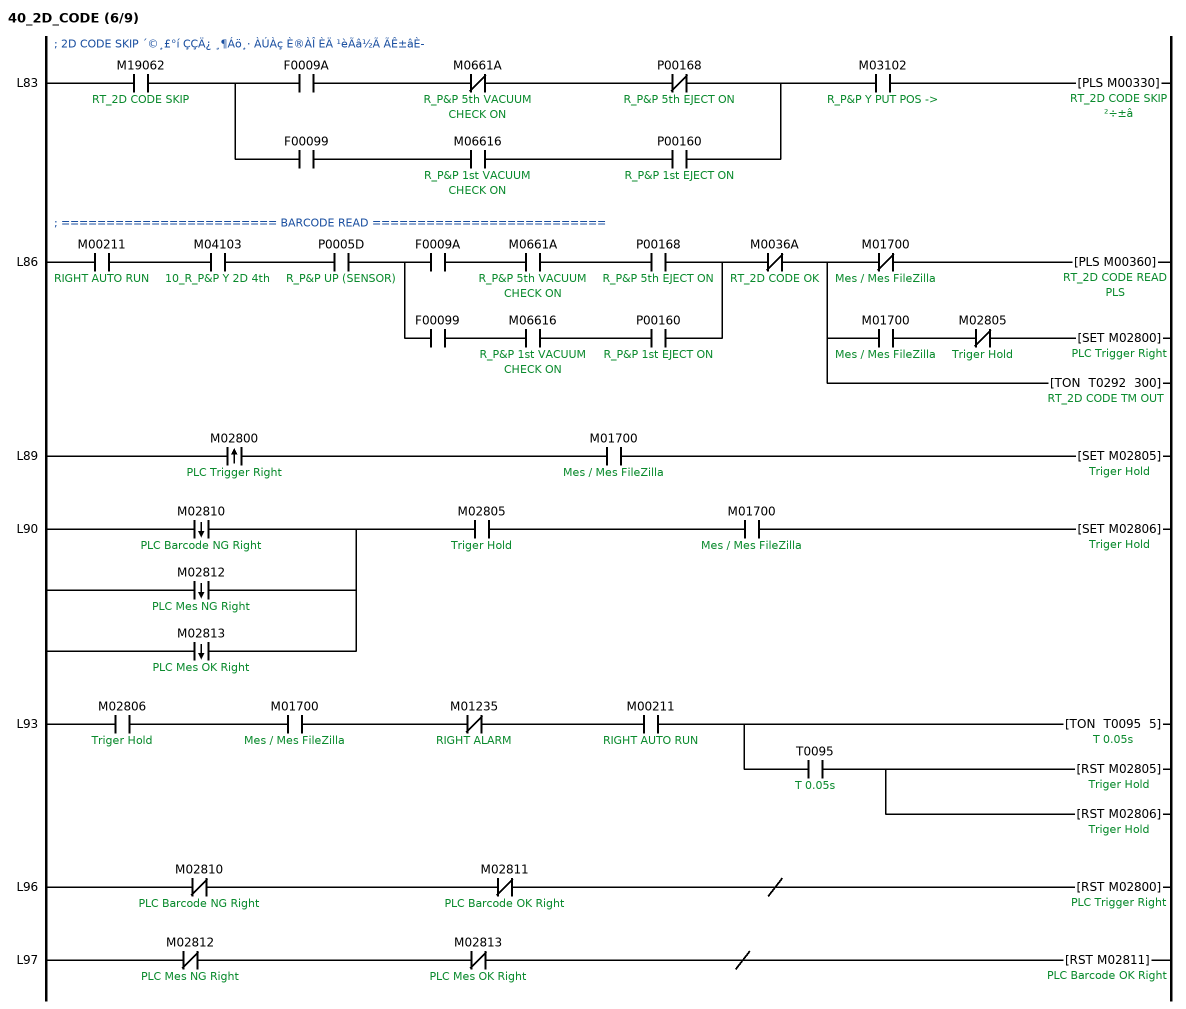
; L83
LOAD      M19062	// RT_2D CODE SKIP
LOAD      F0009A
AND NOT   M0661A	// R_P&P 5th VACUUM CHECK ON
AND NOT   P00168	// R_P&P 5th EJECT ON
LOAD      F00099
AND       M06616	// R_P&P 1st VACUUM CHECK ON
AND       P00160	// R_P&P 1st EJECT ON
OR LOAD
AND LOAD
AND       M03102	// R_P&P Y PUT POS ->
OUTP      M00330	// RT_2D CODE SKIP ²÷±â
// output comment: 2D CODE SKIP ´©¸£°í ÇÇÄ¿ ¸¶Áö¸· ÀÚÀç È®ÀÎ ÈÄ ¹èÃâ½Ã ÃÊ±âÈ­
// ======================== BARCODE READ ==========================
; L86
LOAD      M00211	// RIGHT AUTO RUN
AND       M04103	// 10_R_P&P Y 2D 4th
AND       P0005D	// R_P&P UP (SENSOR)
LOAD      F0009A
AND       M0661A	// R_P&P 5th VACUUM CHECK ON
AND       P00168	// R_P&P 5th EJECT ON
LOAD      F00099
AND       M06616	// R_P&P 1st VACUUM CHECK ON
AND       P00160	// R_P&P 1st EJECT ON
OR LOAD
AND LOAD
AND NOT   M0036A	// RT_2D CODE OK
MPUSH
AND NOT   M01700	// Mes / Mes FileZilla
OUTP      M00360	// RT_2D CODE READ PLS
MLOAD
AND       M01700	// Mes / Mes FileZilla
AND NOT   M02805	// Triger Hold
SET       M02800	// PLC Trigger Right
MPOP
TON       T0292 300	// RT_2D CODE TM OUT
; L89
LOADP     M02800	// PLC Trigger Right
AND       M01700	// Mes / Mes FileZilla
SET       M02805	// Triger Hold
; L90
LOADN     M02810	// PLC Barcode NG Right
ORN       M02812	// PLC Mes NG Right
ORN       M02813	// PLC Mes OK Right
AND       M02805	// Triger Hold
AND       M01700	// Mes / Mes FileZilla
SET       M02806	// Triger Hold
; L93
LOAD      M02806	// Triger Hold
AND       M01700	// Mes / Mes FileZilla
AND NOT   M01235	// RIGHT ALARM
AND       M00211	// RIGHT AUTO RUN
TON       T0095 5	// T 0.05s
AND       T0095	// T 0.05s
RST       M02805	// Triger Hold
RST       M02806	// Triger Hold
; L96
LOAD NOT  M02810	// PLC Barcode NG Right
AND NOT   M02811	// PLC Barcode OK Right
NOT
RST       M02800	// PLC Trigger Right
; L97
LOAD NOT  M02812	// PLC Mes NG Right
AND NOT   M02813	// PLC Mes OK Right
NOT
RST       M02811	// PLC Barcode OK Right

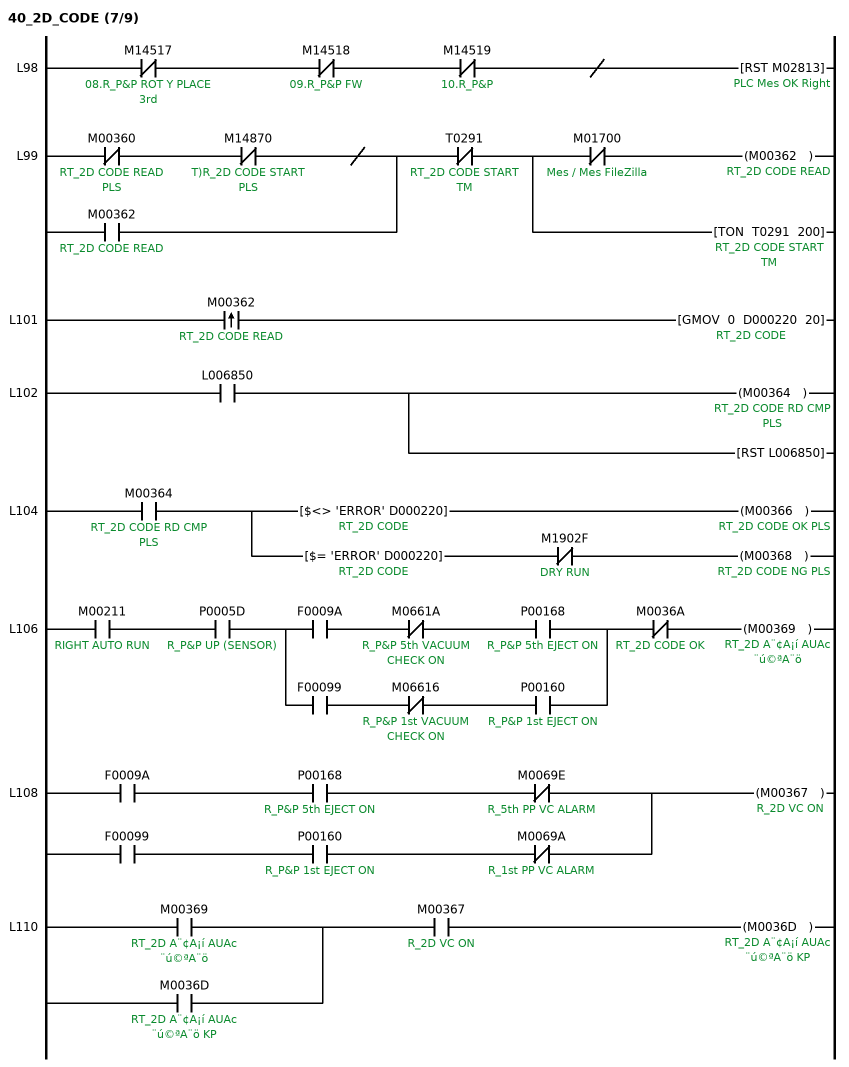
; L98
LOAD NOT  M14517	// 08.R_P&P ROT Y PLACE 3rd
AND NOT   M14518	// 09.R_P&P FW
AND NOT   M14519	// 10.R_P&P
NOT
RST       M02813	// PLC Mes OK Right
; L99
LOAD NOT  M00360	// RT_2D CODE READ PLS
AND NOT   M14870	// T)R_2D CODE START PLS
NOT
OR        M00362	// RT_2D CODE READ
AND NOT   T0291	// RT_2D CODE START TM
MPUSH
AND NOT   M01700	// Mes / Mes FileZilla
OUT       M00362	// RT_2D CODE READ
MPOP
TON       T0291 200	// RT_2D CODE START TM
; L101
LOADP     M00362	// RT_2D CODE READ
GMOV      0 D000220 20	// RT_2D CODE
; L102
LOAD      L006850
OUT       M00364	// RT_2D CODE RD CMP PLS
RST       L006850
; L104
LOAD      M00364	// RT_2D CODE RD CMP PLS
MPUSH
AND$<>    'ERROR' D000220	// RT_2D CODE
OUT       M00366	// RT_2D CODE OK PLS
MPOP
AND$=     'ERROR' D000220	// RT_2D CODE
AND NOT   M1902F	// DRY RUN
OUT       M00368	// RT_2D CODE NG PLS
; L106
LOAD      M00211	// RIGHT AUTO RUN
AND       P0005D	// R_P&P UP (SENSOR)
LOAD      F0009A
AND NOT   M0661A	// R_P&P 5th VACUUM CHECK ON
AND       P00168	// R_P&P 5th EJECT ON
LOAD      F00099
AND NOT   M06616	// R_P&P 1st VACUUM CHECK ON
AND       P00160	// R_P&P 1st EJECT ON
OR LOAD
AND LOAD
AND NOT   M0036A	// RT_2D CODE OK
OUT       M00369	// RT_2D A¨¢A¡í AUAc ¨ú©ªA¨ö
; L108
LOAD      F0009A
AND       P00168	// R_P&P 5th EJECT ON
AND NOT   M0069E	// R_5th PP VC ALARM
LOAD      F00099
AND       P00160	// R_P&P 1st EJECT ON
AND NOT   M0069A	// R_1st PP VC ALARM
OR LOAD
OUT       M00367	// R_2D VC ON
; L110
LOAD      M00369	// RT_2D A¨¢A¡í AUAc ¨ú©ªA¨ö
OR        M0036D	// RT_2D A¨¢A¡í AUAc ¨ú©ªA¨ö KP
AND       M00367	// R_2D VC ON
OUT       M0036D	// RT_2D A¨¢A¡í AUAc ¨ú©ªA¨ö KP

